// TwinCAT 3 PLC project Untitled1
// ProgramVersion: 3.1.4023.0
// CompilerDefines: VISU_USEWSTRING
// libraries:
//   Tc2_Standard, * (Beckhoff Automation GmbH)
//   Tc2_System, * (Beckhoff Automation GmbH)
//   Tc3_Module, * (Beckhoff Automation GmbH)
//   VisuDialogs, * (System)
//   MachineManage,1.3.1.0,Secote
//   VisuSymbols,3.5.10.0,System
// project tree:
//   DUTs/ E_Axis.TcDUT, E_Cylinder.TcDUT, E_LineAxis.TcDUT, E_LoadClose.TcDUT, E_LoadClass.TcDUT, E_MachineType.TcDUT, E_Timer.TcTLEO, ST_TimeOut.TcDUT, E_ProductType.TcDUT, E_Station.TcDUT, ST_Handshake.TcDUT, ST_Input.TcDUT, ST_Output.TcDUT, ST_Recipe.TcDUT, ST_Setting.TcDUT
//   / GlobalTextList.TcGTLO, PlcTask.TcTTO, RecipeManager.TcRMO (not stored), Version.TcPOU, VISU_TASK.TcTTO, 视图管理器.TcVMO (not stored)
//   GVLs/ GVL.TcGVL, GVL_Data.TcGVL, GVL_IO.TcGVL
//   POUs/Device/ ArrayBool_TO_ArrayByte.TcPOU, ArrayBool_TO_Byte.TcPOU, ArrayByte_TO_ArrayBool.TcPOU, Byte_TO_ArrayBool.TcPOU, FB_LineAxis.TcPOU
//   POUs/ MAIN.TcPOU, P_Alarm.TcPOU, P_Device.TcPOU, P_StationAcquire.TcPOU, P_StationLine1Load.TcPOU, P_StationTakeUc.TcPOU, P_StationLine0Buffer.TcPOU, P_StationLine0Load.TcPOU, P_StationOpenLock.TcPOU, P_StationSteering.TcPOU, P_StationTakeUc_M.TcPOU, P_StationUnloadFrock.TcPOU, P_StationUnloadFrock_L.TcPOU, P_StationUnloadUc_L.TcPOU, P_System.TcPOU
//   VISUs/Ctrl/ CtrlAxisInput.TcVIS, CtrlCylinder_Page.TcVIS, CtrlInput.TcVIS (not stored), CtrlLine.TcVIS, CtrlOther.TcVIS (not stored), CtrlOutput.TcVIS, Cyliner1.TcVIS, Cyliner1_1.TcVIS, Cyliner2.TcVIS, Cyliner3.TcVIS, Cyliner4.TcVIS, Cyliner4_1.TcVIS, Cyliner5.TcVIS, FrameMain.TcVIS, ImagePool.TcIPO (not stored), CtrlPageSetting.TcVIS
//   VISUs/ PageData.TcVIS, PageHome.TcVIS, PageMessage.TcVIS, PageMonitor.TcVIS, PageSetting_AcquireLoad.TcVIS, PageSetting_AcquireLoad_2.TcVIS, PageSetting_OpenLock_2.TcVIS, PageSetting_TakeUc.TcVIS, PageSetting_Steering.TcVIS, PageSetting_Other.TcVIS, PageSetting_Unload_L.TcVIS, PageSetting_OpenLock.TcVIS, PageSetting_UnloadFrock.TcVIS, PageSetting_TakeUc_M.TcVIS, PageSetting.TcVIS
//   VISUs/Text/ InputText.TcTLO, LineLoadClose.TcTLO, LineLoadClase.TcTLO, LoadPriority.TcTLO, MachineType.TcTLO, ProductType.TcTLO, ManualText.TcTLO, OutputText.TcTLO, StationName.TcTLO

CONFIGURATION Untitled1
    RESOURCE PLC ON TwinCAT3
        TASK PlcTask(INTERVAL := T#2ms, PRIORITY := 20);
        TASK VISU_TASK(INTERVAL := T#50000us, PRIORITY := 30);
        PROGRAM MAIN WITH PlcTask : MAIN;
        PROGRAM VisuElems_Visu_Prg WITH VISU_TASK : VisuElems.Visu_Prg;
    END_RESOURCE
END_CONFIGURATION

// ---- DUTs/E_Axis.TcDUT
{attribute 'qualified_only'}
{attribute 'strict'}
TYPE E_Axis :
(
	Z := 1// Z轴
);
END_TYPE

// ---- DUTs/E_Cylinder.TcDUT
{attribute 'qualified_only'}
{attribute 'strict'}
TYPE E_Cylinder :
(
Line0Part:=0, //  主流线分料气缸
Line0Prevent, //  主流线阻挡气缸
Line0Push, //  主流线拨料气缸
AcquirePrevent0, //  接驳线前阻挡气缸
AcquirePrevent1, //  接驳线后阻挡气缸
AcquireLift, //  接驳线顶升气缸
AcquirePush, //  接驳模组拨料气缸
AcquireElevator, //  接驳模组升降气缸
SteeringLift, //  转向站顶升气缸
SteeringAcquireElevator, //  转向站接驳升降气缸
SteeringRotate, //  转向站旋转气缸
SteeringAcquireLimit, //  转向站接驳限位气缸
OpenLockPrevent, //  解锁站阻挡气缸
OpenLockLift, //  解锁站顶升气缸
OpenLockPush, //  解锁站侧推气缸
OpenLockRotate, //  解锁站旋转气缸
OpenLockPush2, //  解锁站侧推气缸2
TakeUcPrevent, //  取UC站阻挡气缸
TakeUcLift, //  取UC站顶升气缸
TakeUcPush, //  取UC站侧推气缸
TakeUcRotate, //  取UC站旋转气缸
TakeUcStandard, //  取UC站校平气缸
UnloadFrockPrevent, //  下工装站阻挡气缸
UnloadFrockLift, //  下工装站顶升气缸
UnloadFrockPush, //  下工装站拨料气缸
TakeUc1Y, //  取UC模组平移Y气缸
TakeUc1Z1, //  取UC模组升降Z1气缸
TakeUc1Z2, //  取UC模组升降Z2气缸
TakeUc1Rotate, //  取UC模组旋转气缸
TakeUc1Clamp, //  取UC模组夹紧气缸
UnloadUcElevator, //  下UC皮带升降气缸
UnloadUcConveyorPush, //  下UC皮带拨料气缸
UnloadFrockConveyorPrevent, //  下工装皮带升降气缸
UnloadFrockConveyorPush, //  下工装皮带拨料气缸
OpenLockElevator,// 解锁站升降气缸
OpenLockPin,// 解锁站压紧气缸
TakeUcElevator,// 取UC站升降气缸
TakeUcPush1,// 取UC站侧推气缸1
UnloadUcBeltTipper,// 下UC皮带翻转
UnloadUcBeltLift,// 下UC皮带顶升
OpenLockTranslation,// 解锁站解锁平移气缸
TakeUcFrockClamp,//取UC站工装夹紧气缸
OpenLockPressPush,//解锁站解压侧推气缸
OpenLockPressRotate,//解锁站解压旋转气缸
AcquirePrevent2,//  接驳线前前阻挡气缸
Line0PushElevator, //  主流线拨料升降气缸
Length
);
END_TYPE

// ---- DUTs/E_LineAxis.TcDUT
{attribute 'qualified_only'}
{attribute 'strict'}
TYPE E_LineAxis :
(
	UnloadUc := 1,// 下Uc线体
	UnloadForck,// 下工装线条
	Acquire,// 接驳站线体
	Dismantling,// 拆解站线体
	AcquireFront // 接驳站前线体
);
END_TYPE

// ---- DUTs/E_LoadClose.TcDUT
{attribute 'qualified_only'}
{attribute 'strict'}
TYPE E_LoadClose :
(
	None:=0,
	Line0,// 关闭Line0
	Acquire// 关闭接驳站上料
);
END_TYPE

// ---- DUTs/E_LoadClass.TcDUT
{attribute 'qualified_only'}
{attribute 'strict'}
TYPE E_LoadClass :
(
	None:=0,
	Line0,// 优先Line0
	Acquire,// 优先接驳站
	Sensor // 优先传感器检测
);
END_TYPE

// ---- DUTs/E_MachineType.TcDUT
{attribute 'qualified_only'}
{attribute 'strict'}
TYPE E_MachineType :
(
	None:=0,
	_367,
	_200,
	_373,
	_069,
	_311
);
END_TYPE

// ---- DUTs/E_Timer.TcTLEO
{attribute 'qualified_only'}
{attribute 'strict'}
TYPE E_Timer :
(
	Timer0 := 0,
	Line0PriorityOnDelay,     // 主流线优先置位延时
	Line0PriorityOffDelay,    // 主流线优先复位延时
	SteeringCheck1F,
	OpenLockCheckF,
	Timer5,
	Timer6,
	Timer7,
	Timer8,
	Timer9,
	Timer10,
	Timer11,
	Timer12,
	Timer13,
	Timer14,
	Timer15,
	Timer16,
	Timer17,
	Timer18,
	Timer19
	
);
END_TYPE

// ---- DUTs/ST_TimeOut.TcDUT
TYPE ST_TimeOut :
STRUCT
	bAcquireCheck2:             BOOL;//接驳线光电检测超时
    bLine0Check3:               BOOL;//主流线到位光电检测超时	
	bOpenLockCheck:             BOOL;//解锁站到位光电检测超时
	bSteeringCheck1:            BOOL;//转向站到位光电检测超时
	bTakeUcCheck1:              BOOL;//取UC站到位光电检测超时
	bUnloadUcCheck1:			BOOL;//翻转气缸到位光电检测超时
	bUnloadFrockCheck1:         BOOL;//下工装站到位光电检测超时
	bUnloadFrockConveyorCheck2: BOOL;//下工装皮带到位光电检测超时
	bUnloadUcCheck2:            BOOL;//下UC皮带到位光电检测超时
	bLine0Check2:               BOOL;//主流线阻挡光电检测超时
	bLine0PushElevatorUp:       BOOL;//主流线拨料升降气缸上升速度过慢
END_STRUCT
END_TYPE

// ---- DUTs/E_ProductType.TcDUT
{attribute 'qualified_only'}
{attribute 'strict'}
TYPE E_ProductType :
(
	None:= 0,
	Left,
	Right
);
END_TYPE

// ---- DUTs/E_Station.TcDUT
{attribute 'qualified_only'}
{attribute 'strict'}
TYPE E_Station :
(
Acquire:=0,//接驳站
Line0Buffer,//主流线缓存
Line0Load,//主流线上料
OpenLock,//解锁站
Steering,//转向站
TakeUc,//取Uc站
TakeUc_M,//取Uc模组
UnloadFrock,//下工装
UnloadFrock_L,//下工装线体
UnloadUc_L,//下UC线体
Line1Load,//接驳线上料
Length
);
END_TYPE

// ---- DUTs/ST_Handshake.TcDUT
TYPE ST_Handshake :
STRUCT
	bBufferToLoad:				BOOL;// 上料缓存站 请求 上料站 放料
	bLoadToBuffer:				BOOL;// 上料站 收到 缓存站请求
	
	bLine1ToAcquire:			BOOL;// 接驳线 请求 接驳站 收料
	bAcquireToLine1:			BOOL;// 接驳站 收到 接驳线请求
	
	bBufferToAcquire:			BOOL;// 上料缓存站 请求 接驳站收料
	bAcquireToBuffer:			BOOL;// 接驳站收 上料缓存站请求
	
	bSteering:					BOOL;// 转向站 请求 放料
	bSteeringOk:				BOOL;// 收到 转向站请求信号
	
	bOpenToSteering:			BOOL;// 解锁站 请求 转向站放料
	bSteeringToOpen:			BOOL;// 转向站 收到 解锁站请求
	
	bTakeUcToOpen:				BOOL;// 取U站 请求 解锁站放料
	bOpenToTakeUc:				BOOL;// 解锁站 收到 取Uc站请求
	
	bTakeUcToTakeUc_M:			BOOL;// 取UC站 请求 取UC模组取料
	bTakeUc_MToTakeUc:			BOOL;// 取Uc模组 收到取Uc站请求
	
	bTakeUcToTakeUc_M_2:			BOOL;// 取UC站 请求 取UC模组取料
	bTakeUc_MToTakeUc_2:			BOOL;// 取Uc模组 收到取Uc站请求
	
	
	bUnloadFrockToTakeUc:		BOOL;//	下工装站 请求 取Uc站放料
	bTakeUcToUnloadFrock:		BOOL;// 取Uc站 收到 下工装站请求
	
	bTakeUc_MToUnloadUcConveyor:BOOL;// 下Uc模组 请求 下Uc线体放料
	bUnloadUcConveyorToTakeUc_M:BOOL;// 下Uc线体 收到 下Uc模组请求
	
	bUnloadFrockToUnloadFrock_L:BOOL;// 下工装站 请求 下工装线体放料
	bUnloadFrock_LToUnloadFrock:BOOL;// 下工装线体 收到 下工装站请求   
END_STRUCT
END_TYPE

// ---- DUTs/ST_Input.TcDUT
TYPE ST_Input :
STRUCT
bStart:BOOL;//启动 IN00
bStop:bool;//停止 IN01
bResetAlarm:bool;//复位 IN02
bEStop:bool;//急停 IN03
bDoor:bool;//安全门开关 IN04
bFrockCloseCheck:BOOL;//工装误合盖检测 IN05
bOpenLockCheck0:BOOL;//解锁站流入光电 IN06
bNone3:bool;//预留 IN07
bLine0PushElevator_Cyl_H:BOOL;//主流线拨料升降气缸原位 IN08
bLine0PushElevator_Cyl_W:BOOL;//主流线拨料升降气缸工作位 IN09
bNone6:bool;//预留 IN0A
bNone7:bool;//预留 IN0B
bLine0Push_Cyl_Safe:BOOL;//主流线拨料气缸安全位 IN0C
bAcquireCheck0:BOOL;//接驳线前阻挡光电 IN0D
bAcquirePrevent2_Cyl_H:BOOL;//接驳线前前阻挡气缸原位 IN0E
bAcquirePrevent2_Cyl_W:BOOL;//接驳线前前阻挡气缸工作位 IN0F
bLine0Part_Cyl_H:bool;//主流线分料气缸原位 IN10
bLine0Part_Cyl_W:bool;//主流线分料气缸工作位 IN11
bLine0Prevent_Cyl_H:bool;//主流线阻挡气缸原位 IN12
bLine0Prevent_Cyl_W:bool;//主流线阻挡气缸工作位 IN13
bLine0Push_Cyl_H:bool;//主流线拨料气缸原位 IN14
bLine0Push_Cyl_W:bool;//主流线拨料气缸工作位 IN15
bAcquirePrevent0_Cyl_H:bool;//接驳线前阻挡气缸原位 IN16
bAcquirePrevent0_Cyl_W:bool;//接驳线前阻挡气缸工作位 IN17
bAcquirePrevent1_Cyl_H:bool;//接驳线后阻挡气缸原位 IN18
bAcquirePrevent1_Cyl_W:bool;//接驳线后阻挡气缸工作位 IN19
bAcquireLift_Cyl_H:bool;//接驳线顶升气缸原位 IN1A
bAcquireLift_Cyl_W:bool;//接驳线顶升气缸工作位 IN1B
bAcquirePush_Cyl_H:bool;//接驳模组拨料气缸原位 IN1C
bAcquirePush_Cyl_W:bool;//接驳模组拨料气缸工作位 IN1D
bAcquireElevator_Cyl_H:bool;//接驳模组升降气缸原位 IN1E
bAcquireElevator_Cyl_W:bool;//接驳模组升降气缸工作位 IN1F
bSteeringLift_Cyl_H:bool;//转向站顶升气缸原位 IN20
bSteeringLift_Cyl_W:bool;//转向站顶升气缸工作位 IN21
bSteeringAcquireElevator_Cyl_H:bool;//转向站接驳升降气缸原位 IN22
bSteeringAcquireElevator_Cyl_W:bool;//转向站接驳升降气缸工作位 IN23
bSteeringRotate_Cyl_H:bool;//转向站旋转气缸原位 IN24
bSteeringRotate_Cyl_W:bool;//转向站旋转气缸工作位 IN25
bSteeringAcquireLimit_Cyl_H:bool;//转向站接驳限位气缸原位 IN26
bSteeringAcquireLimit_Cyl_W:bool;//转向站接驳限位气缸工作位 IN27
bOpenLockPrevent_Cyl_H:bool;//解锁站阻挡气缸原位 IN28
bOpenLockPrevent_Cyl_W:bool;//解锁站阻挡气缸工作位 IN29
bOpenLockLift_Cyl_H:bool;//解锁站顶升气缸原位 IN2A
bOpenLockLift_Cyl_W:bool;//解锁站顶升气缸工作位 IN2B
bOpenLockPush_Cyl_H:bool;//解锁站侧推气缸原位 IN2C
bOpenLockPush_Cyl_W:bool;//解锁站侧推气缸工作位 IN2D
bOpenLockRotate_Cyl_H:bool;//解锁站旋转气缸原位 IN2E
bOpenLockRotate_Cyl_W:bool;//解锁站旋转气缸工作位 IN2F
bOpenLockPush2_Cyl_H:bool;//解锁站侧推气缸2原位 IN30
bOpenLockPush2_Cyl_W:bool;//解锁站侧推气缸2工作位 IN31
bTakeUcPrevent_Cyl_H:bool;//取UC站阻挡气缸原位 IN32
bTakeUcPrevent_Cyl_W:bool;//取UC站阻挡气缸工作位 IN33
bTakeUcLift_Cyl_H:bool;//取UC站顶升气缸原位 IN34
bTakeUcLift_Cyl_W:bool;//取UC站顶升气缸工作位 IN35
bTakeUcPush_Cyl_H:bool;//取UC站侧推气缸原位 IN36
bTakeUcPush_Cyl_W:bool;//取UC站侧推气缸工作位 IN37
bTakeUcRotate_Cyl_H:bool;//取UC站旋转气缸原位 IN38
bTakeUcRotate_Cyl_W:bool;//取UC站旋转气缸工作位 IN39
bTakeUcStandard_Cyl_H:bool;//取UC站校平气缸原位 IN3A
bTakeUcStandard_Cyl_W:bool;//取UC站校平气缸工作位 IN3B
bTakeUcFrockClamp_Cyl_H:BOOL;//取UC站工装夹紧气缸原位 IN3C
bTakeUcFrockClamp_Cyl_W:BOOL;//取UC站工装夹紧气缸工作位 IN3D
bUnloadFrockPrevent_Cyl_H:bool;//下工装站阻挡气缸原位 IN3E
bUnloadFrockPrevent_Cyl_W:bool;//下工装站阻挡气缸工作位 IN3F
bUnloadFrockLift_Cyl_H:bool;//下工装站顶升气缸原位 IN40
bUnloadFrockLift_Cyl_W:bool;//下工装站顶升气缸工作位 IN41
bUnloadFrockPush_Cyl_H:bool;//下工装站拨料气缸原位 IN42
bUnloadFrockPush_Cyl_W:bool;//下工装站拨料气缸工作位 IN43
bTakeUc1Y_Cyl_H:bool;//取UC模组平移Y气缸原位 IN44
bTakeUc1Y_Cyl_W:bool;//取UC模组平移Y气缸工作位 IN45
bTakeUc1Z1_Cyl_H:bool;//取UC模组升降Z1气缸原位 IN46
bTakeUc1Z1_Cyl_W:bool;//取UC模组升降Z1气缸工作位 IN47
bTakeUc1Z2_Cyl_H:bool;//取UC模组升降Z2气缸原位 IN48
bTakeUc1Z2_Cyl_W:bool;//取UC模组升降Z2气缸工作位 IN49
bTakeUc1Rotate_Cyl_H:bool;//取UC模组旋转气缸原位 IN4A
bTakeUc1Rotate_Cyl_W:bool;//取UC模组旋转气缸工作位 IN4B
bTakeUc1Clamp_Cyl_H:bool;//取UC模组夹紧气缸原位 IN4C
bTakeUc1Clamp_Cyl_W:bool;//取UC模组夹紧气缸工作位 IN4D
bUnloadUcElevator_Cyl_H:bool;//下UC皮带升降气缸原位 IN4E
bUnloadUcElevator_Cyl_W:bool;//下UC皮带升降气缸工作位 IN4F
bUnloadUcConveyorPush_Cyl_H:bool;//下UC皮带拨料气缸原位 IN50
bUnloadUcConveyorPush_Cyl_W:bool;//下UC皮带拨料气缸工作位 IN51
bUnloadFrockConveyorPrevent_Cyl_H:bool;//下工装皮带升降气缸原位 IN52
bUnloadFrockConveyorPrevent_Cyl_W:bool;//下工装皮带升降气缸工作位 IN53
bUnloadFrockConveyorPush_Cyl_H:bool;//下工装皮带拨料气缸原位 IN54
bUnloadFrockConveyorPush_Cyl_W:bool;//下工装皮带拨料气缸工作位 IN55
bOpenLockPressPush_Cyl_H:BOOL;//解锁站解压侧推气缸原位 IN56
bOpenLockPressPush_Cyl_W:BOOL;//解锁站解压侧推气缸工作位 IN57
bOpenLockPressRotate_Cyl_H:BOOL;//解锁站解压旋转气缸原位 IN58
bOpenLockPressRotate_Cyl_W:BOOL;//解锁站解压旋转气缸工作位 IN59
bNone34:bool;//预留 IN5A
bNone35:bool;//预留 IN5B
bUnloadUcBeltTipper_Cyl_H:bool;//下UC皮带翻转气缸缩回 IN5C
bUnloadUcBeltTipper_Cyl_W:bool;//下UC皮带翻转气缸伸出 IN5D
bUnloadUcBeltLift_Cyl_H:bool;//下UC皮带顶升气缸缩回 IN5E
bUnloadUcBeltLift_Cyl_W:bool;//下UC皮带顶升气缸伸出 IN5F
bLine0Check1:bool;//主流线分料光电 IN60
bLine0Check2:bool;//主流线阻挡光电 IN61
bLine0Check3:bool;//主流线到位光电 IN62
bAcquireCheck1:bool;//接驳线流入光电 IN63
bAcquireCheck2:bool;//接驳线到位光电 IN64
bSteeringCheck1:bool;//转向站到位光电 IN65
bOpenLockCheck:bool;//解锁站到位光电 IN66
bTakeUcCheck1:bool;//取UC站到位光电 IN67
bUnloadFrockCheck1:bool;//下工装站到位光电 IN68
bUnloadUcCheck1:bool;//下UC皮带流入光电 IN69
bUnloadUcCheck2:bool;//下UC皮带到位光电 IN6A
bUnloadFrockCheck0:BOOL;//下工装站流入光电 IN6B
bUnloadFrockConveyorCheck2:bool;//下工装皮带到位光电 IN6C
bUnloadUcBeltTipper:bool;//下uc皮带翻转光电 IN6D
bTakeUcCheck0:BOOL;//取UC站流入光电 IN6E
bTakeUc1Y_Cyl_Safe:BOOL;//取UC模组平移Y气缸安全位 IN6F
bOpenLockElevator_Cyl_H:bool;//解锁站升降气缸原位 IN70
bOpenLockElevator_Cyl_W:bool;//解锁站升降气缸工作位 IN71
bOpenLockTranslation_Cyl_H:bool;//解锁站解锁平移原位 IN72
bOpenLockTranslation_Cyl_W:bool;//解锁站解锁平移工作位 IN73
bOpenLockPin_Cyl_H:bool;//解锁站按压气缸到原位 IN74
bOpenLockPin_Cyl_W:bool;//解锁站按压气缸到工作位 IN75
bTakeUcElevator_Cyl_H:bool;//取UC站升降气缸原位 IN76
bTakeUcElevator_Cyl_W:bool;//取UC站升降气缸工作位 IN77
bTakeUcPush1_Cyl_H:bool;//取UC站侧推1气缸到原位 IN78
bTakeUcPush1_Cyl_W:bool;//取UC站侧推1气缸到工作位 IN79
bNone45:bool;//预留 IN7A
bNone46:bool;//预留 IN7B
bNone47:bool;//预留 IN7C
bNone48:bool;//预留 IN7D
bNone49:bool;//预留 IN7E
bNone50:bool;//预留 IN7F

END_STRUCT
END_TYPE

// ---- DUTs/ST_Output.TcDUT
TYPE ST_Output :
STRUCT
bBeacon_Red:BOOL;//三色灯红 OUT00
bBeacon_Yellow:bool;//三色灯黄 OUT01
bBeacon_Green:bool;//三色灯绿 OUT02
bBeacon_Buzzer:bool;//蜂鸣器 OUT03
bRuning:bool;//运行指示灯 OUT04
bStop:bool;//停止指示灯 OUT05
bLED:bool;//照明灯 OUT06
bNone1:bool;//预留 OUT07
bOpenLockPressPush_Cyl_H:BOOL;//解锁站解压侧推气缸到原位 OUT08
bOpenLockPressPush_Cyl_W:BOOL;//解锁站解压侧推气缸到工作位 OUT09
bOpenLockPressRotate_Cyl_H:BOOL;//解锁站解压旋转气缸到原位 OUT0A
bOpenLockPressRotate_Cyl_W:BOOL;//解锁站解压旋转气缸到工作位 OUT0B
bLine0PushElevator_Cyl_H:BOOL;//主流线拨料升降气缸到原位 OUT0C
bLine0PushElevator_Cyl_W:BOOL;//主流线拨料升降气缸到工作位 OUT0D
bAcquirePrevent2_Cyl_H:BOOL;//接驳线前前阻挡气缸缩回 OUT0E
bAcquirePrevent2_Cyl_W:BOOL;//接驳线前前阻挡气缸伸出 OUT0F
bLine0Part_Cyl_H:bool;//主流线分料气缸缩回 OUT10
bLine0Part_Cyl_W:bool;//主流线分料气缸伸出 OUT11
bLine0Prevent_Cyl_H:bool;//主流线阻挡气缸缩回 OUT12
bLine0Prevent_Cyl_W:bool;//主流线阻挡气缸伸出 OUT13
bLine0Push_Cyl_H:bool;//主流线拨料气缸缩回 OUT14
bLine0Push_Cyl_W:bool;//主流线拨料气缸伸出 OUT15
bAcquirePrevent0_Cyl_H:bool;//接驳线前阻挡气缸缩回 OUT16
bAcquirePrevent0_Cyl_W:bool;//接驳线前阻挡气缸伸出 OUT17
bAcquirePrevent1_Cyl_H:bool;//接驳线后阻挡气缸缩回 OUT18
bAcquirePrevent1_Cyl_W:bool;//接驳线后阻挡气缸伸出 OUT19
bAcquireLift_Cyl_H:bool;//接驳线顶升气缸缩回 OUT1A
bAcquireLift_Cyl_W:bool;//接驳线顶升气缸伸出 OUT1B
bAcquirePush_Cyl_H:bool;//接驳模组拨料气缸缩回 OUT1C
bAcquirePush_Cyl_W:bool;//接驳模组拨料气缸伸出 OUT1D
bAcquireElevator_Cyl_H:bool;//接驳模组升降气缸缩回 OUT1E
bAcquireElevator_Cyl_W:bool;//接驳模组升降气缸伸出 OUT1F
bSteeringLift_Cyl_H:bool;//转向站顶升气缸缩回 OUT20
bSteeringLift_Cyl_W:bool;//转向站顶升气缸伸出 OUT21
bSteeringAcquireElevator_Cyl_H:bool;//转向站接驳升降气缸缩回 OUT22
bSteeringAcquireElevator_Cyl_W:bool;//转向站接驳升降气缸伸出 OUT23
bSteeringRotate_Cyl_H:bool;//转向站旋转气缸缩回 OUT24
bSteeringRotate_Cyl_W:bool;//转向站旋转气缸伸出 OUT25
bSteeringAcquireLimit_Cyl_H:bool;//转向站接驳限位气缸缩回 OUT26
bSteeringAcquireLimit_Cyl_W:bool;//转向站接驳限位气缸伸出 OUT27
bOpenLockPrevent_Cyl_H:bool;//解锁站阻挡气缸缩回 OUT28
bOpenLockPrevent_Cyl_W:bool;//解锁站阻挡气缸伸出 OUT29
bOpenLockLift_Cyl_H:bool;//解锁站顶升气缸缩回 OUT2A
bOpenLockLift_Cyl_W:bool;//解锁站顶升气缸伸出 OUT2B
bOpenLockPush_Cyl_H:bool;//解锁站侧推气缸缩回 OUT2C
bOpenLockPush_Cyl_W:bool;//解锁站侧推气缸伸出 OUT2D
bOpenLockRotate_Cyl_H:bool;//解锁站旋转气缸缩回 OUT2E
bOpenLockRotate_Cyl_W:bool;//解锁站旋转气缸伸出 OUT2F
bOpenLockPush2_Cyl_H:bool;//解锁站侧推气缸2缩回 OUT30
bOpenLockPush2_Cyl_W:bool;//解锁站侧推气缸2伸出 OUT31
bTakeUcPrevent_Cyl_H:bool;//取UC站阻挡气缸缩回 OUT32
bTakeUcPrevent_Cyl_W:bool;//取UC站阻挡气缸伸出 OUT33
bTakeUcLift_Cyl_H:bool;//取UC站顶升气缸缩回 OUT34
bTakeUcLift_Cyl_W:bool;//取UC站顶升气缸伸出 OUT35
bTakeUcPush_Cyl_H:bool;//取UC站侧推气缸缩回 OUT36
bTakeUcPush_Cyl_W:bool;//取UC站侧推气缸伸出 OUT37
bTakeUcRotate_Cyl_H:bool;//取UC站旋转气缸缩回 OUT38
bTakeUcRotate_Cyl_W:bool;//取UC站旋转气缸伸出 OUT39
bTakeUcStandard_Cyl_H:bool;//取UC站校平气缸原位 OUT3A
bTakeUcStandard_Cyl_W:bool;//取UC站校平气缸工作位 OUT3B
bTakeUcFrockClamp_Cyl_H:BOOL;//取UC站工装夹紧气缸原位 OUT3C
bTakeUcFrockClamp_Cyl_W:bool;//取UC站工装夹紧气缸工作位 OUT3D
bUnloadFrockPrevent_Cyl_H:BOOL;//下工装站阻挡气缸缩回 OUT3E
bUnloadFrockPrevent_Cyl_W:bool;//下工装站阻挡气缸伸出 OUT3F
bUnloadFrockLift_Cyl_H:bool;//下工装站顶升气缸缩回 OUT40
bUnloadFrockLift_Cyl_W:bool;//下工装站顶升气缸伸出 OUT41
bUnloadFrockPush_Cyl_H:bool;//下工装站拨料气缸缩回 OUT42
bUnloadFrockPush_Cyl_W:bool;//下工装站拨料气缸伸出 OUT43
bTakeUc1Y_Cyl_H:bool;//取UC模组平移Y气缸缩回 OUT44
bTakeUc1Y_Cyl_W:bool;//取UC模组平移Y气缸伸出 OUT45
bTakeUc1Z1_Cyl_H:bool;//取UC模组升降Z1气缸缩回 OUT46
bTakeUc1Z1_Cyl_W:bool;//取UC模组升降Z1气缸伸出 OUT47
bTakeUc1Z2_Cyl_H:bool;//取UC模组升降Z2气缸缩回 OUT48
bTakeUc1Z2_Cyl_W:bool;//取UC模组升降Z2气缸伸出 OUT49
bTakeUc1Rotate_Cyl_H:bool;//取UC模组旋转气缸缩回 OUT4A
bTakeUc1Rotate_Cyl_W:bool;//取UC模组旋转气缸伸出 OUT4B
bTakeUc1Clamp_Cyl_H:bool;//取UC模组夹紧气缸缩回 OUT4C
bTakeUc1Clamp_Cyl_W:bool;//取UC模组夹紧气缸伸出 OUT4D
bUnloadUcElevator_Cyl_H:bool;//下UC皮带升降气缸缩回 OUT4E
bUnloadUcElevator_Cyl_W:bool;//下UC皮带升降气缸伸出 OUT4F
bUnloadUcConveyorPush_Cyl_H:bool;//下UC皮带拨料气缸缩回 OUT50
bUnloadUcConveyorPush_Cyl_W:bool;//下UC皮带拨料气缸伸出 OUT51
bUnloadFrockConveyorPrevent_Cyl_H:bool;//下工装皮带升降气缸缩回 OUT52
bUnloadFrockConveyorPrevent_Cyl_W:bool;//下工装皮带升降气缸伸出 OUT53
bUnloadFrockConveyorPush_Cyl_H:bool;//下工装皮带拨料气缸缩回 OUT54
bUnloadFrockConveyorPush_Cyl_W:bool;//下工装皮带拨料气缸伸出 OUT55
bAcquireFrontAxis:BOOL;//接驳站前步进 OUT56
bAcquireAxis:bool;//接驳线步进 OUT57
bDismantlingAxis:bool;//拆解线步进 OUT58
bUnloadUcAxis:bool;//下UC皮带步进 OUT59
bUnloadFrock:bool;//下工装皮带步进 OUT5A
bNone21:bool;//预留 OUT5B
bUnloadUcBeltTipper_Cyl_H:bool;//下UC皮带翻转气缸缩回 OUT5C
bUnloadUcBeltTipper_Cyl_W:bool;//下UC皮带翻转气缸伸出 OUT5D
bUnloadUcBeltLift_Cyl_H:bool;//下UC皮带顶升气缸缩回 OUT5E
bUnloadUcBeltLift_Cyl_W:bool;//下UC皮带顶升气缸伸出 OUT5F
bOpenLockElevator_Cyl_H:bool;//解锁站升降气缸原位 OUT60
bOpenLockElevator_Cyl_W:bool;//解锁站升降气缸工作位 OUT61
bOpenLockTranslation_Cyl_H:bool;//解锁站解锁平移原位 OUT62
bOpenLockTranslation_Cyl_W:bool;//解锁站解锁平移工作位 OUT63
bOpenLockPin_Cyl_H:bool;//解锁站按压气缸到原位 OUT64
bOpenLockPin_Cyl_W:bool;//解锁站按压气缸到工作位 OUT65
bTakeUcElevator_Cyl_H:bool;//取UC站升降气缸原位 OUT66
bTakeUcElevator_Cyl_W:bool;//取UC站升降气缸工作位 OUT67
bTakeUcPush1_Cyl_H:bool;//取UC站侧推1气缸到原位 OUT68
bTakeUcPush1_Cyl_W:bool;//取UC站侧推1气缸到工作位 OUT69
bNone35:BOOL;//预留 OUT6A
bNone36:BOOL;//预留 OUT6B
bNone37:BOOL;//预留 OUT6C
bNone38:BOOL;//预留 OUT6D
bNone39:bool;//预留 OUT6E
bNone40:bool;//预留 OUT6F

END_STRUCT
END_TYPE

// ---- DUTs/ST_Recipe.TcDUT
TYPE ST_Recipe :
STRUCT
	arrInputTon:				ARRAY[0..7,0..15] OF UINT;
	arrOutputTon:				ARRAY[0..6,0..15] OF UINT;
	arrAutoTon:				    ARRAY[0..19] OF UINT;	
	
	eMachineType:				E_MachineType;
	eProductType:               E_ProductType;//产品类型（左，右）
	eLoadClass:					E_LoadClass;
	eLoadClose:					E_LoadClose;
	
	bLuxshardict:				BOOL;
END_STRUCT
END_TYPE

// ---- DUTs/ST_Setting.TcDUT
TYPE ST_Setting :
STRUCT
	bDryRun:					BOOL;// 空跑
	bManualLoad:				BOOL;// 手动上料
	bManualUnloadUc:			BOOL;// 手动下UC
	bManualUnloadFrock:			BOOL;// 手动下工装
	arrStationShield:			ARRAY[0..20] OF BOOL;// 工站使能信号
	bLine0BufferShield:         BOOL;// 主流分料屏蔽
	bSafeDoorShield:            BOOL;// 安全门屏蔽
	bOpenLockPressShield:       BOOL;// 解锁站解除保压屏蔽
	bAcquirePrevent2Shield:     BOOL;// 接驳线前前阻挡气缸屏蔽
	bStopFrontStation:          BOOL;// 不允许前站放料
	bLine0Priority:             BOOL;// 优先主流线上料
	bFrockCloseCheckShield:     BOOL;// 工装误合盖检测屏蔽
END_STRUCT
END_TYPE

// ---- GVLs/GVL.TcGVL
{attribute 'qualified_only'}
VAR_GLOBAL
	I:					ST_Input;
	Q:					ST_Output;
	stSetting:			ST_Setting;// 设置参数
	
	stShield_I:			ARRAY[0..7,0..15] OF  BOOL;
	stShield_Q:			ARRAY[0..6,0..15] OF  BOOL;
	
	stHandshake:		ST_Handshake;
				
	arrFbLine:			ARRAY[0..10] OF FB_LineAxis;// 流线控制
	
    stOverTime:			ST_TimeOut;//光电超时报警 
	
	_arrAutoTimer:		ARRAY[0..19] OF  TON;//自动流程延时 
	_arrAutoTimerOut:	ARRAY[0..19] OF  BOOL;//自动流程延时输出
	
	TakeUcSafeCheckNG_OpenLock:  BOOL;	//解锁站工装误合盖检测NG记忆
	TakeUcSafeCheckNG_TakeUc:  BOOL;    //取UC站读取解锁站工装误合盖检测NG记忆
	AlarmResetMark:     BOOL;           //311机型主流线拨料升降气缸上升速度过慢报警复位标记
	
END_VAR

// ---- GVLs/GVL_Data.TcGVL
{attribute 'qualified_only'}
VAR_GLOBAL PERSISTENT
	stRecipe:					ST_Recipe;// 配方文件
END_VAR

// ---- GVLs/GVL_IO.TcGVL
{attribute 'qualified_only'}
VAR_GLOBAL
	I_Temp :				ARRAY[0..7,0..15] OF  BOOL;//由绝对点位的字节数组 转化成的布尔数组
	Q_Temp :				ARRAY[0..6,0..15] OF  BOOL;//由绝对点位的字节数组 转化成的布尔数组
	
	I AT %I*:				ARRAY[0..15] OF BYTE;//绝对点位 输入
	Q AT %Q*:				ARRAY[0..13] OF BYTE;//绝对点位 输出

	EIP_I_ConnState AT %I*:				UDINT;// 输入
	EIP_I_Var4090   AT %I*:				WORD;// 输入	
	EIP_Q_ConnCtrl  AT %Q*:				UDINT;// 输出
	EIP_Q_Var4091   AT %Q*:				WORD;// 输出	
	
	
	AxisInput AT %I*:		UDINT;			
END_VAR

// ---- POUs/MAIN.TcPOU
PROGRAM MAIN
VAR
	VERSION:STRING;
END_VAR

GVL_Data.stRecipe.bLuxshardict:=TRUE;

VERSION:='5.5.0';
P_System();
P_Alarm();
P_Device();

P_StationAcquire();// 接驳站
P_StationLine0Buffer();// Line0上料缓存站
P_StationLine0Load();// Line0上料站
P_StationOpenLock();// 解锁站
P_StationSteering();// 转向站
P_StationTakeUc();// 取UC
P_StationTakeUc_M();// 取UC模组
P_StationUnloadFrock();// 下工装
P_StationUnloadFrock_L();// 下工装线条
P_StationUnloadUc_L();// 下UC线条
P_StationLine1Load();// Line1上料站


IF GVL_Data.stRecipe.eMachineType=E_MachineType._367 THEN
	GVL_IO.EIP_Q_Var4091.1:=GVL_P.G_stSystem.stMode.bAutoRunning AND NOT GVL.I.bLine0Check1 AND  NOT GVL.stSetting.bStopFrontStation;//给前站设备要料信号
ELSE
	GVL_IO.EIP_Q_Var4091.1:=GVL_P.G_stSystem.stMode.bAutoRunning AND NOT GVL.I.bAcquireCheck0 AND  NOT GVL.stSetting.bStopFrontStation;//给前站设备要料信号
END_IF

END_PROGRAM

// ---- Version.TcPOU
PROGRAM Version
VAR
END_VAR

//	版本号		修改人		修改日期		修改内容
//	1.2.0		李天		2021.06.27		311空跑后优化373解锁校平气缸
//	1.3.0		李天		2021.06.27		添加下工装阻挡气缸判断
//  1.4.0      刘雪峰       2021.06.28      添加下工装阻挡气缸屏蔽，优化气缸屏蔽，增加气缸空跑程序的调用选择
//  1.5.0      刘雪峰       2021.06.28      添加轴命名，添加取UC模组升降Z2气缸IO屏蔽，增加版本号界面显示，完善转向站和取uc模组流程，增加取uc模组z1z2气缸控制方法调用的判断,完善各机型气缸空跑程序
//  2.0.0      刘雪峰       2021.06.29      更新IO,气缸、轴excel,新增取UC工装夹紧气缸和IO,更新input和output结构体,更新E_cycliner枚举变量,按照机型屏蔽新增的气缸和IO,更新input和output的Textlist,优化取UC工站和取UC模组工站流程,完善正常模式下调用的A_Cylinder程序
//  2.1.0      刘雪峰       2021.07.01      更新气缸调试部分的界面程序，增加产品类型选择，优化转向站和下UC线体流程，添加取UC模组夹紧气缸工作位和解锁站侧推气缸2初始位在空跑时的屏蔽
//	2.2.0		李天		2021.07.02		修改373解锁校平气缸2动作,该气缸只需一直伸出即可;
//  2.2.1      刘雪峰       2021.07.05      修改部分气缸的界面调试控件，优化转向站初始化气缸动作流程；
//  2.3.0       王恒        2021.07.14      增加拨料站（Switch）和翻转站（Tipper）,将接驳模组拨料气缸和接驳模组升降气缸单独组成拨料站，将下UC皮带翻转气缸和下UC皮带顶升气缸单独组成翻转站;
//  2.3.1       王恒        2021.07.23      增加各工站到位光电检测超时报警;增加气缸界面按工站分页功能;主界面增加界面CT显示;增加生产计数显示;增加各到位光电信号显示;增加从转向站手动上料和从下UC、下工装皮带末端手动下料功能；增加屏蔽取UC模组功能，使投入工装时，只验证解锁与扣合，不验证夹取UC动作；
//                                          增加初始化检测各工站光电是否检测有料功能，并在初始化结束添加再次提醒操作员人工检查的5级报警;201机型下UC皮带流入光电IN6B代替下UC皮带翻转光电IN6D,用来检测UC是否到位，下UC皮带翻转光电IN6D不再使用；因为取UC模组Z1气缸上升速度较慢，所以下调了取UC模组Z1气缸的上限位，使Z1气缸的行程尽可能减少;
//  2.3.2       李天        2021.07.25      增加伺服轴持续接触极限报警，无法点动脱离问题，增加相应指示灯和复位功能；
//	2.4.0		李天		2021.07.26		将王恒新增的两个工站（接驳模组站及下UC线体旋转站） 再改回去
//	2.5.0		李天		2021.07.26		在RH069中待料测试 并修改一些细节 不影响整体流程
//	2.5.1		李天		2021.07.27		将手动下UC 手动下工装 手动上料 开放到界面
//	2.5.2		李天		2021.07.27		将报警显示控件放大
//	2.6.0		李天		2021.07.27		修改手动上料跳转空步号问题
//	2.6.1		李天		2021.07.28		添加用户权限 用户名：Admin 密码：333
//	2.6.2		李伟3		2021.07.28		优化201取UC站侧推气缸动作 可提前推出
//	2.7.0		李天		2021.07.31		将下UC流线及下工装流线到位光电报警等级改成3级
//	2.7.1		李伟3		2021.08.2		将自动流程中1471步中取UC模组平移Y气缸硬件IO修改为气缸功能块状态位
//	3.0.0		李伟3		2021.08.3		1.将自动流程中1471步中取UC模组平移Y气缸气缸功能块状态位修改为硬件IO
//                                          2.暂时取消手动页面权限管理，方便调试
//                                          3.将IO监控页面IN6B下工装线体流入光电变更为下工装流线流入光电
//                                          4.修改取UC模组自动程序，添加分支:设备机型为311时，取UC旋转气缸不旋转放料
//                                          5.将设备内工位检测到位光电传感器超时报警由五级报警提升为三级报警，并修复报警无法复位问题
//                                          6.添加 IN6F取UC模组平移Y气缸安全位 传感器,并修改动作流程
//                                          7.修改和优化了311机型设备 取UC站&取UC模组 的自动动作流程,缩短CT时间
//                                          8.在自动程序中添加 下UC线体到位检测超时 报警
//	3.0.1		李伟3		2021.08.5		1.屏蔽画面中添加屏蔽主流线分料气缸的功能
//                                          2.将主画面计数清零按钮增加用户权限
//                                          3.优化修改367机型 取UC模组 自动流程,缩短CT
//                                          4.优化画面按钮相关中文显示
//                                          5.修复了下工装站初始化撞机的问题
//	3.0.2		李伟3		2021.08.6		1.屏蔽画面中添加 蜂鸣器屏蔽 和 安全门屏蔽 的功能
//                                          2.增加 设备运行中安全门被打开 报警
//	4.0.0		李伟3		2021.08.12		1.373机型解锁站增加两个气缸，增加手动&自动&初始化程序
//                                          2.修复373机型手动画面校平气缸未屏蔽的问题
//                                          3.修复373机型IO画面未使用IO点没有屏蔽的问题
//                                          4.修复设备蜂鸣器响声不正常的问题
//                                          5.优化367机型取UC站的自动流程
//	4.1.0		李伟3		2021.08.13		1.增加接驳线阻挡气缸&接驳线光电传感器，增加手动&自动&初始化程序
//	4.1.1		李伟3		2021.08.16		1.优化不同机型手动页面&IO监控页面的显示问题
//	4.2.0		李伟3		2021.08.24		1.将新加的接驳站前流水线由急停按钮控制改为继电器控制，增加手自动程序
//	4.2.1		李伟3		2021.08.25		1.优化201机型下UC皮带翻转顶升气缸动作流程，先让顶升气缸上升再放UC，防止损伤排线
//	4.2.2		李伟3		2021.08.31		1.优化主流线分料气缸和阻挡气缸的动作逻辑,修改主流线分料气缸缩回端为原位,增加主流线阻挡光电检测超时报警
//	4.3.0		李伟3		2021.09.02		1.367机型增加主流线拨料升降气缸，修改手自动程序及画面
//                                          2.修改取UC站初始化动作流程，修复367机型取UC站初始化异常的问题
//	5.0.0		李伟3		2021.09.07		1.增加通过EIP与前站信号交互的配置和程序
//                                          2.修改主流线到位光电检测超时时间为20S,因为主流线速度过慢会误引发报警
//	5.1.0		李伟3		2021.09.10		1.优化了主流线和接驳线上料优先级选择部分的程序，画面上增加了优先级下拉菜单选择
//                                          2.画面上增加了停止前站放料的按钮
//                                          3.增加 主流线拨料气缸安全位 IN0C 传感器，优化367主流线上料流程
//                                          4.增加主流线与接驳线上料优先级根据传感器自动切换逻辑
//                                          5.优化与前站交互要料逻辑
//	5.2.0		李伟3		2021.09.16		1.311机型增加检测工装误合盖传感器，修改动作流程及画面
//                                          2.367机型增加解锁站流入光电传感器，优化动作流程，缩短CT
//                                          3.373机型增加取UC站流入光电传感器，优化动作流程，缩短CT
//                                          4.373机型增加主流线传感器,优化367机型主流线拨料气缸动作，增加主流线拨料升降气缸上升速度过慢报警，防止损伤产品
//                                          5.优化自动程序中所使用的延时，画面上增加延时时间设置
//                                          6.将打开安全门由一级报警修改为3级报警，方便维护
//                                          7.修复取UC站初始化时与取UC模组撞机的问题
//	5.3.0		李伟3		2021.09.17		1.373机型取UC站增加检测工装误合盖传感器，修改动作流程及画面
//	5.4.0		李伟3		2021.09.17		1.修改解锁站和取UC站的放料逻辑，缩短CT
//	5.5.0		李伟3		2021.09.17		1.将接驳站分料气缸和阻挡气缸分离为单独工站，优化交互逻辑

END_PROGRAM

// ---- POUs/P_System.TcPOU
PROGRAM P_System
VAR
	_arrFbButton:			ARRAY[0..10] OF FB_Button;
	_arrTon:				ARRAY[0..10] OF TON;
	_fbCT:					FB_CycleTime1;
	_cttime:				REAL;
	
	_rTRIG:					R_TRIG;
	_iProductionCount:      INT;//产能计数
	_bCountZero:			BOOL;//产能计数清零
END_VAR

A_Machine();
A_System();

ACTION A_Machine:
//CT测试
_fbCT(Execute:=G_arrCylinder[E_Cylinder.TakeUcLift].stOutput.bWork, CycleTime=> );
_cttime:=TIME_TO_REAL(_fbCT.CycleTime)/1000;
//复位 退出空跑模式
IF G_stSystem.stInput.bReset THEN
	GVL.stSetting.bDryRun:=FALSE;
END_IF

//产能计数
_rTRIG(CLK:= G_arrCylinder[E_Cylinder.OpenLockLift].stOutput.bWork, Q=> );
IF G_stSystem.stMode.bAutoRunning AND NOT GVL.stSetting.bDryRun AND _rTRIG.Q THEN
	_iProductionCount:=_iProductionCount+1;
END_IF
IF NOT G_stSystem.stMode.bAutoRunning  AND  _bCountZero THEN
	_iProductionCount:=0;
END_IF
END_ACTION

ACTION A_System:
G_stSystem.stInput.bEStop:=NOT GVL.I.bEStop;
_arrTon[0](IN:=GVL.I.bResetAlarm,PT:=T#3S , Q=>G_stSystem.stInput.bInit , ET=> );


GVL.Q.bBeacon_Buzzer:=G_stSystem.stOutput.bLightRed AND NOT MachineManage.G_stSystem.stInput.bQuiet;
GVL.Q.bRuning:=GVL.Q.bBeacon_Green:=G_stSystem.stOutput.bLightGreen;
GVL.Q.bStop:=GVL.Q.bBeacon_Red:=G_stSystem.stOutput.bLightRed;
GVL.Q.bBeacon_Yellow:=G_stSystem.stOutput.bLightYellow;

_arrFbButton[0](In:=G_stSystem.stInput.bStart, CLK:=GVL.I.bStart );
_arrFbButton[1](In:= G_stSystem.stInput.bStop, CLK:=GVL.I.bStop );
_arrFbButton[2](In:=G_stSystem.stInput.bResetAlarm , CLK:= GVL.I.bResetAlarm  );

G_stSystem.stLogConfig.bExecute:=TRUE;
G_stSystem.stLogConfig.sFilePath:='D:\PLC\Log\System';

P_Machine(StationCount:=E_Station.Length);
END_ACTION

END_PROGRAM

// ---- POUs/P_Alarm.TcPOU
PROGRAM P_Alarm
VAR
	_arrFbErrorTag1:				ARRAY[0..20] OF  FB_ErrorTag;
	_arrFbErrorTag2:				ARRAY[0..20] OF  FB_ErrorTag;
	_arrFbErrorTag3:				ARRAY[0..20] OF  FB_ErrorTag;
	_arrFbErrorTag4:				ARRAY[0..20] OF  FB_ErrorTag;
	_arrFbErrorTag5:				ARRAY[0..20] OF  FB_ErrorTag;
	
	_i:								INT;
	
	_bFirstRun:						BOOL:=true;
END_VAR

G_stError.bSaveLog:=TRUE;
G_stError.sFileLogPath:='D:\PLC\Log\Error';

A_Alarm1();
A_Alarm2();
A_Alarm3();
A_Alarm4();
A_Alarm5();

ACTION A_Alarm1:

_i:=0;
_arrFbErrorTag1[_i].Enable:=NOT GVL.I.bEStop;
_arrFbErrorTag1[_i].Language[E_Language.Chinese]:="急停被按下";


_i:=1;
_arrFbErrorTag1[_i].Enable:=GVL_Data.stRecipe.eMachineType=E_MachineType.None;
_arrFbErrorTag1[_i].Language[E_Language.Chinese]:="设备类型未选择";

_i:=2;
_arrFbErrorTag1[_i].Enable:=GVL_Data.stRecipe.eProductType=E_ProductType.None;
_arrFbErrorTag1[_i].Language[E_Language.Chinese]:="产品类型未选择";



FOR _i:=0 TO 20 BY 1 DO
_arrFbErrorTag1[_i](
	System:=G_stSystem , 
	Error:=G_stError , 
	ID:=TO_BYTE(_i+50) , 
	Category:=E_ErrorCategory.Safety , 
	InfoIndex:= , 
	Enable:= , 
	Message:= , 
	Level:=1 , 
	Position:="P_Alarm:A_Alarm1" , 
	ErrorTime:= , 
	Language:= , 
	Erroring=> , 
	ErrorCode=> );
END_FOR
END_ACTION

ACTION A_Alarm2:
_i:=0;
_arrFbErrorTag2[_i].Enable:=G_arrCylinder[E_Cylinder.TakeUc1Clamp].stOutput.bWork AND NOT G_stSystem.stMode.bHomeDone;
_arrFbErrorTag2[_i].Language[E_Language.Chinese]:="请将夹紧气缸松开后再初始化";


FOR _i:=0 TO 20 BY 1 DO
_arrFbErrorTag2[_i](
	System:=G_stSystem , 
	Error:=G_stError , 
	ID:=TO_BYTE(52) , 
	Category:=E_ErrorCategory.Other , 
	InfoIndex:=TO_BYTE(_i) , 
	Enable:= , 
	Message:= , 
	Level:=2 , 
	Position:="P_Alarm:A_Alarm2" , 
	ErrorTime:= , 
	Language:= , 
	Erroring=> , 
	ErrorCode=> );
END_FOR
END_ACTION

ACTION A_Alarm3:
_i:=0;
_arrFbErrorTag3[_i].Enable:=(G_stSystem.stMode.bHomeDone AND G_arrStation[E_Station.OpenLock].iStepNow = 1000) 
AND (GVL_IO.I_Temp[6,4](*接驳线到位光电*) OR GVL_IO.I_Temp[6,2](*主流线到位光电*) OR GVL_IO.I_Temp[6,6](*解锁站到位光电*) OR 
GVL_IO.I_Temp[6,5](*转向站到位光电*) OR GVL_IO.I_Temp[6,7](*取UC站到位光电*) OR GVL_IO.I_Temp[6,8](*下工装站到位光电*) OR GVL_IO.I_Temp[6,10](*下UC皮带到位光电*) OR GVL_IO.I_Temp[6,12](*下工装皮带到位光电*)) ;
_arrFbErrorTag3[_i].Language[E_Language.Chinese]:="机台中有残余物料，请手动清料";
_arrFbErrorTag3[_i].Language[E_Language.English]:="There is a residue in the machine. Please clean the material manually";

_i:=1;
_arrFbErrorTag3[_i].ErrorTime:=T#5S;
_arrFbErrorTag3[_i].Enable:=GVL.stOverTime.bAcquireCheck2 AND GVL_P.G_stSystem.stMode.bAutoRunning;
_arrFbErrorTag3[_i].Language[E_Language.Chinese]:="接驳线光电检测超时";
_arrFbErrorTag3[_i].Language[E_Language.English]:="Relay line photoelectric detection timeout";

_i:=2;
_arrFbErrorTag3[_i].ErrorTime:=T#20S;
_arrFbErrorTag3[_i].Enable:=GVL.stOverTime.bLine0Check3 AND GVL_P.G_stSystem.stMode.bAutoRunning;
_arrFbErrorTag3[_i].Language[E_Language.Chinese]:="主流线到位光电检测超时";
_arrFbErrorTag3[_i].Language[E_Language.English]:="The mainstream line is in place to photoelectric test timeout";

_i:=3;
_arrFbErrorTag3[_i].ErrorTime:=T#5S;
_arrFbErrorTag3[_i].Enable:=GVL.stOverTime.bLine0Check2 AND GVL_P.G_stSystem.stMode.bAutoRunning;
_arrFbErrorTag3[_i].Language[E_Language.Chinese]:="主流线阻挡光电检测超时";
_arrFbErrorTag3[_i].Language[E_Language.English]:="The main line blocks the photoelectric detection timeout";

_i:=4;
_arrFbErrorTag3[_i].ErrorTime:=T#5S;
_arrFbErrorTag3[_i].Enable:=GVL.stOverTime.bUnloadFrockConveyorCheck2 AND GVL_P.G_stSystem.stMode.bAutoRunning;
_arrFbErrorTag3[_i].Language[E_Language.Chinese]:="下工装皮带到位光电检测超时";
_arrFbErrorTag3[_i].Language[E_Language.English]:="The next working belt is in the photoelectric detection timeout";

_i:=5;
_arrFbErrorTag3[_i].ErrorTime:=T#5S;
_arrFbErrorTag3[_i].Enable:=GVL.stOverTime.bUnloadUcCheck2 AND GVL_P.G_stSystem.stMode.bAutoRunning;
_arrFbErrorTag3[_i].Language[E_Language.Chinese]:="下UC皮带到位光电检测超时";
_arrFbErrorTag3[_i].Language[E_Language.English]:="The lower uc belt is in place to photoelectric test timeout";

_i:=6;
_arrFbErrorTag3[_i].ErrorTime:=T#5S;
_arrFbErrorTag3[_i].Enable:=NOT P_StationSteering._bManual AND GVL.stOverTime.bOpenLockCheck AND GVL_P.G_stSystem.stMode.bAutoRunning;
_arrFbErrorTag3[_i].Language[E_Language.Chinese]:="解锁站到位光电检测超时";
_arrFbErrorTag3[_i].Language[E_Language.English]:="The solution lock station is in place for photoelectric detection timeout";

_i:=7;
_arrFbErrorTag3[_i].ErrorTime:=T#5S;
_arrFbErrorTag3[_i].Enable:=GVL.stOverTime.bSteeringCheck1 AND GVL_P.G_stSystem.stMode.bAutoRunning;
_arrFbErrorTag3[_i].Language[E_Language.Chinese]:="转向站到位光电检测超时";
_arrFbErrorTag3[_i].Language[E_Language.English]:="Turn to the station to photoelectric test timeout";

_i:=8;
_arrFbErrorTag3[_i].ErrorTime:=T#5S;
_arrFbErrorTag3[_i].Enable:=GVL.stOverTime.bTakeUcCheck1 AND GVL_P.G_stSystem.stMode.bAutoRunning;
_arrFbErrorTag3[_i].Language[E_Language.Chinese]:="取UC站到位光电检测超时";
_arrFbErrorTag3[_i].Language[E_Language.English]:="The uc station is in place for photoelectric detection timeout";

_i:=9;
_arrFbErrorTag3[_i].ErrorTime:=T#5S;
_arrFbErrorTag3[_i].Enable:=GVL.stOverTime.bUnloadUcCheck1 AND GVL_P.G_stSystem.stMode.bAutoRunning;
_arrFbErrorTag3[_i].Language[E_Language.Chinese]:="翻转气缸到位光电检测超时";
_arrFbErrorTag3[_i].Language[E_Language.English]:="The inverted cylinder is in place for photoelectric detection timeout";

_i:=10;
_arrFbErrorTag3[_i].ErrorTime:=T#5S;
_arrFbErrorTag3[_i].Enable:=GVL.stOverTime.bUnloadFrockCheck1 AND GVL_P.G_stSystem.stMode.bAutoRunning;
_arrFbErrorTag3[_i].Language[E_Language.Chinese]:="下工装站到位光电检测超时";
_arrFbErrorTag3[_i].Language[E_Language.English]:="The next working station is in place for photoelectric detection timeout";

_i:=11;
_arrFbErrorTag3[_i].ErrorTime:=T#5S;
_arrFbErrorTag3[_i].Enable:=G_arrStation[E_Station.OpenLock].iStepNow=1100 AND GVL.I.bLine0Check1 AND NOT GVL.I.bLine0Check2 AND GVL_P.G_stSystem.stMode.bAutoRunning;
_arrFbErrorTag3[_i].Language[E_Language.Chinese]:="IN61 主流线阻挡光电检测超时";
_arrFbErrorTag3[_i].Language[E_Language.English]:="The IN61 Line0Check2 detection timeout";

_i:=12;
_arrFbErrorTag3[_i].ErrorTime:=T#0S;
_arrFbErrorTag3[_i].Enable:=GVL.stOverTime.bLine0PushElevatorUp AND GVL_P.G_stSystem.stMode.bAutoRunning;
_arrFbErrorTag3[_i].Language[E_Language.Chinese]:="拨料升降气缸上升速度过慢报警";
_arrFbErrorTag3[_i].Language[E_Language.English]:="The IN61 Line0Check2 detection timeout";

_i:=13;
_arrFbErrorTag3[_i].ErrorTime:=T#0S;
_arrFbErrorTag3[_i].Enable:=NOT GVL.I.bDoor AND GVL_P.G_stSystem.stMode.bAutoRunning AND NOT GVL.stSetting.bSafeDoorShield;
_arrFbErrorTag3[_i].Language[E_Language.Chinese]:="设备运行中安全门被打开";
_arrFbErrorTag3[_i].Language[E_Language.English]:="Safe door open in running";


(*_i:=10;
_arrFbErrorTag3[_i].Enable:=NOT GVL.I.bDoor;
_arrFbErrorTag3[_i].Language[E_Language.Chinese]:="安全门打开";*)

IF gvl_p.G_stSystem.stInput.bResetAlarm THEN
	GVL.stOverTime.bAcquireCheck2:=FALSE;
	GVL.stOverTime.bLine0Check2:=FALSE;
	GVL.stOverTime.bOpenLockCheck:=FALSE;
	GVL.stOverTime.bSteeringCheck1:=FALSE;
	GVL.stOverTime.bTakeUcCheck1:=FALSE;
	GVL.stOverTime.bUnloadFrockCheck1:=FALSE;
	GVL.stOverTime.bUnloadFrockConveyorCheck2:=FALSE;
	GVL.stOverTime.bUnloadUcCheck1:=FALSE;
	GVL.stOverTime.bUnloadUcCheck2:=FALSE;
	IF GVL.stOverTime.bLine0PushElevatorUp THEN
		GVL.stOverTime.bLine0PushElevatorUp:=FALSE;
		GVL.AlarmResetMark:=TRUE;
	END_IF
END_IF

FOR _i:=0 TO 20 BY 1 DO
_arrFbErrorTag3[_i](
	System:=G_stSystem , 
	Error:=G_stError , 
	ID:=TO_BYTE(53) , 
	Category:=E_ErrorCategory.Other , 
	InfoIndex:=TO_BYTE(_i) , 
	Enable:= , 
	Message:= , 
	Level:=3 , 
	Position:="P_Alarm:A_Alarm3" , 
	ErrorTime:= , 
	Language:= , 
	Erroring=> , 
	ErrorCode=> );
END_FOR
END_ACTION

ACTION A_Alarm4:








FOR _i:=0 TO 20 BY 1 DO
_arrFbErrorTag4[_i](
	System:=G_stSystem , 
	Error:=G_stError , 
	ID:=TO_BYTE(54) , 
	Category:=E_ErrorCategory.Other , 
	InfoIndex:=TO_BYTE(_i) , 
	Enable:= , 
	Message:= , 
	Level:=4 , 
	Position:="P_Alarm:A_Alarm4" , 
	ErrorTime:= , 
	Language:= , 
	Erroring=> , 
	ErrorCode=> );
END_FOR
END_ACTION

ACTION A_Alarm5:
_i:=0;
_arrFbErrorTag5[_i].Enable:=(G_stSystem.stMode.bHomeDone AND G_arrStation[E_Station.OpenLock].iStepNow = 1000) ;
_arrFbErrorTag5[_i].Language[E_Language.Chinese]:="请确认机台是否有残余物料,点击启动继续流程";
_arrFbErrorTag5[_i].Language[E_Language.English]:="Please confirm whether there is any residual material . Click the start continue process";

//_i:=1;
//_arrFbErrorTag5[_i].ErrorTime:=T#5S;
//_arrFbErrorTag5[_i].Enable:=NOT P_StationSteering._bManual AND GVL.stOverTime.bOpenLockCheck;
//_arrFbErrorTag5[_i].Language[E_Language.Chinese]:="解锁站到位光电检测超时";
//_arrFbErrorTag5[_i].Language[E_Language.English]:="The solution lock station is in place for photoelectric detection timeout";

//_i:=2;
//_arrFbErrorTag5[_i].ErrorTime:=T#5S;
//_arrFbErrorTag5[_i].Enable:=GVL.stOverTime.bSteeringCheck1;
//_arrFbErrorTag5[_i].Language[E_Language.Chinese]:="转向站到位光电检测超时";
//_arrFbErrorTag5[_i].Language[E_Language.English]:="Turn to the station to photoelectric test timeout";

//_i:=3;
//_arrFbErrorTag5[_i].ErrorTime:=T#5S;
//_arrFbErrorTag5[_i].Enable:=GVL.stOverTime.bTakeUcCheck1;
//_arrFbErrorTag5[_i].Language[E_Language.Chinese]:="取UC站到位光电检测超时";
//_arrFbErrorTag5[_i].Language[E_Language.English]:="The uc station is in place for photoelectric detection timeout";

//_i:=4;
//_arrFbErrorTag5[_i].ErrorTime:=T#5S;
//_arrFbErrorTag5[_i].Enable:=GVL.stOverTime.bUnloadUcCheck1;
//_arrFbErrorTag5[_i].Language[E_Language.Chinese]:="翻转气缸到位光电检测超时";
//_arrFbErrorTag5[_i].Language[E_Language.English]:="The inverted cylinder is in place for photoelectric detection timeout";

//_i:=5;
//_arrFbErrorTag5[_i].ErrorTime:=T#5S;
//_arrFbErrorTag5[_i].Enable:=GVL.stOverTime.bUnloadFrockCheck1;
//_arrFbErrorTag5[_i].Language[E_Language.Chinese]:="下工装站到位光电检测超时";
//_arrFbErrorTag5[_i].Language[E_Language.English]:="The next working station is in place for photoelectric detection timeout";



FOR _i:=0 TO 20 BY 1 DO
_arrFbErrorTag5[_i](
	System:=G_stSystem , 
	Error:=G_stError , 
	ID:=TO_BYTE(55) , 
	Category:=E_ErrorCategory.Other , 
	InfoIndex:=TO_BYTE(_i) , 
	Enable:= , 
	Message:= , 
	Level:=5 , 
	Position:="P_Alarm:A_Alarm5" , 
	ErrorTime:= , 
	Language:= , 
	Erroring=> , 
	ErrorCode=> );
END_FOR
END_ACTION

END_PROGRAM

// ---- POUs/P_StationSteering.TcPOU
PROGRAM P_StationSteering
VAR
	_station:					REFERENCE TO ST_SystemStation;
	
	_arrTemp:					ARRAY[0..10] OF BOOL;
	_bEnable: 					BOOL;
	
	_bManual:                   BOOL;//  手动上料

END_VAR

_station REF= G_arrStation[E_Station.Steering];
_station.arrName[E_Language.Chinese]:="转向站";
_station.arrName[E_Language.Vietnamese]:="Quay về vị trí";
_bEnable:=NOT GVL.stSetting.arrStationShield[E_Station.Steering];
A_Home();
A_Auto();

_bManual:=GVL.stSetting.bManualLoad ;

ACTION A_Auto:
CASE _station.iStepNow OF
	1000:
		_station.arrInfo[E_Language.Chinese]:="初始化完成等待启动";
		IF  _bEnable THEN
			_station.iStepNext:=1101;
		END_IF
	1101:
		_station.arrInfo[E_Language.Chinese]:="判断是否有料";
		IF NOT GVL.I.bSteeringCheck1 THEN
			_station.iStepNext:=SEL(_bManual,1201,1551);
		END_IF
	1201:
		_station.arrInfo[E_Language.Chinese]:="请求放料";
		GVL.stHandshake.bSteering:=TRUE;
		IF GVL.stHandshake.bSteeringOk THEN
			_station.iStepNext:=1301;
		END_IF
	1301:
	     _station.arrInfo[E_Language.Chinese]:="检测物料是否到转向站";
		 GVL.stOverTime.bSteeringCheck1:=TRUE;
	    IF GVL.I.bSteeringCheck1 THEN
			GVL.stOverTime.bSteeringCheck1:=FALSE;
			_station.iStepNext:=1311;
		END_IF
	1311:
		_station.arrInfo[E_Language.Chinese]:="复位放料请求";
		GVL.stHandshake.bSteering:=FALSE;
		IF NOT  GVL.stHandshake.bSteeringOk THEN
			_station.iStepNext:=1351;
		END_IF
	1351:
		_station.arrInfo[E_Language.Chinese]:="限位气缸缩回";
		IF  G_arrFbCylinder[E_Cylinder.SteeringAcquireLimit].M_HomeRequest() THEN
			_station.iStepNext:=1401;
		END_IF
	1401:
		_station.arrInfo[E_Language.Chinese]:="顶升气缸伸出";
		IF M_LiftWork() THEN
			_station.iStepNext:=1451;
	    END_IF
	1451:
		_station.arrInfo[E_Language.Chinese]:="接驳升降气缸缩回";
		CASE GVL_Data.stRecipe.eMachineType OF
			E_MachineType._367:
				IF  G_arrFbCylinder[E_Cylinder.SteeringAcquireElevator].M_HomeRequest() THEN
					_station.iStepNext:=1501;
		    	END_IF
			ELSE
				_station.iStepNext:=1501;
		END_CASE
	1501:
		_station.arrInfo[E_Language.Chinese]:="旋转气缸动作";
		IF M_RotateWork() THEN
			_station.iStepNext:=1551;
		END_IF
	1551:
		_station.arrInfo[E_Language.Chinese]:="等待解锁站请求放料";
		IF GVL.stHandshake.bOpenToSteering THEN
			GVL.stHandshake.bSteeringToOpen:=TRUE;
			_station.iStepNext:=SEL(_bManual,1561,1651);
		END_IF
	1561:
		_station.arrInfo[E_Language.Chinese]:="接驳升降气缸缩回";
        IF  G_arrFbCylinder[E_Cylinder.SteeringAcquireElevator].M_HomeRequest() THEN
			_station.iStepNext:=1601;
		END_IF
	1601:
		_station.arrInfo[E_Language.Chinese]:="顶升气缸缩回";
		IF M_LiftHome() THEN
			_station.iStepNext:=1651;
		END_IF
	1651:
		_station.arrInfo[E_Language.Chinese]:="等待复位放料请求";
		IF NOT GVL.stHandshake.bOpenToSteering THEN
			GVL.stHandshake.bSteeringToOpen:=FALSE;
			_station.iStepNext:=SEL(_bManual,1655,1101);
		END_IF
	1655:
		CASE GVL_Data.stRecipe.eMachineType OF
			E_MachineType._311:
				_station.iStepNext:=1661;
			E_MachineType._367:	
				GVL.stHandshake.bSteering:=TRUE;
				_station.iStepNext:=1701;		
			ELSE
				_station.iStepNext:=1701;
		END_CASE
	1661:
		_station.arrInfo[E_Language.Chinese]:="顶升气缸伸出";
		IF M_LiftWork() THEN
			_station.iStepNext:=1671;
		END_IF
	1671:
		_station.arrInfo[E_Language.Chinese]:="旋转气缸复位";
		IF M_RotateHome() THEN
			_station.iStepNext:=1681;
		END_IF
	1681:
		_station.arrInfo[E_Language.Chinese]:="顶升气缸缩回";
		IF M_LiftHome() THEN
			_station.iStepNext:=1701;
		END_IF
	1701:
		_station.arrInfo[E_Language.Chinese]:="接驳升降气缸伸出 限位气缸伸出";
		IF G_arrFbCylinder[E_Cylinder.SteeringAcquireElevator].M_WorkRequest() and G_arrFbCylinder[E_Cylinder.SteeringAcquireLimit].M_WorkRequest() THEN
			_station.iStepNext:=1901;
		END_IF
	1901:
		_station.arrInfo[E_Language.Chinese]:="旋转气缸复位"; 
		IF M_RotateHome() THEN
			_station.iStepNext:=SEL(GVL_Data.stRecipe.eMachineType=E_MachineType._367,1101,1201);
		END_IF
END_CASE
END_ACTION

ACTION A_Home:
CASE _station.iStepNow OF
	0:
		_station.arrInfo[E_Language.Chinese]:="等待初始化";
		_station.iStepNext:=SEL(_bEnable,1000,100);
	100:
	    IF GVL_Data.stRecipe.eMachineType = E_MachineType._367 THEN
			_station.iStepNext:=150;
			ELSE
				_station.iStepNext:=450;
		END_IF
	150:
		_station.arrInfo[E_Language.Chinese]:="顶升气缸伸出";
		    IF G_arrFbCylinder[E_Cylinder.SteeringLift].M_WorkRequest() THEN
		     	_station.iStepNext:=200;
		    END_IF
		
	200:
		_station.arrInfo[E_Language.Chinese]:="接驳升降气缸缩回";
		IF G_arrFbCylinder[E_Cylinder.SteeringAcquireElevator].M_HomeRequest()  THEN
			_station.iStepNext:=300;
		END_IF
	
	300:
		_station.arrInfo[E_Language.Chinese]:="旋转气缸复位";
		IF G_arrFbCylinder[E_Cylinder.SteeringRotate].M_HomeRequest() THEN
			_station.iStepNext:=400;
		END_IF
	400:
		_station.arrInfo[E_Language.Chinese]:="顶升气缸缩回";
		IF G_arrFbCylinder[E_Cylinder.SteeringLift].M_HomeRequest() THEN
			_station.iStepNext:=450;
		END_IF
	450:
		IF NOT _bManual THEN
			_station.iStepNext:=500;
		ELSE
			_station.iStepNext:=700;
		END_IF
	500:
		_station.arrInfo[E_Language.Chinese]:="接驳升降气缸伸出";
		IF G_arrFbCylinder[E_Cylinder.SteeringAcquireElevator].M_WorkRequest()  THEN
			_station.iStepNext:=600;
		END_IF
	600:
		_station.arrInfo[E_Language.Chinese]:="限位气缸伸出";
		IF  G_arrFbCylinder[E_Cylinder.SteeringAcquireLimit].M_WorkRequest() THEN
			_station.iStepNext:=1000;
		END_IF
		
		
	700:
	    _station.arrInfo[E_Language.Chinese]:="接驳升降气缸缩回";
		IF G_arrFbCylinder[E_Cylinder.SteeringAcquireElevator].M_HomeRequest()  THEN
			_station.iStepNext:=800;
		END_IF
	800:
	    _station.arrInfo[E_Language.Chinese]:="限位气缸缩回";
		IF  G_arrFbCylinder[E_Cylinder.SteeringAcquireLimit].M_HomeRequest() THEN
			_station.iStepNext:=1000;
		END_IF
		
	
END_CASE
END_ACTION

METHOD M_LiftHome : BOOL
VAR_INPUT
END_VAR
CASE GVL_Data.stRecipe.eMachineType OF
	E_MachineType._367:
		M_LiftHome:=G_arrFbCylinder[E_Cylinder.SteeringLift].M_HomeRequest();
	ELSE
		M_LiftHome:=TRUE;		
END_CASE
END_METHOD

METHOD M_LiftWork : BOOL
VAR_INPUT
END_VAR
CASE GVL_Data.stRecipe.eMachineType OF
	E_MachineType._367:	
		M_LiftWork:=G_arrFbCylinder[E_Cylinder.SteeringLift].M_WorkRequest();
	ELSE
		M_LiftWork:=TRUE;
END_CASE
END_METHOD

METHOD M_RotateHome : BOOL
VAR_INPUT
END_VAR
CASE GVL_Data.stRecipe.eMachineType OF
	E_MachineType._367:
		M_RotateHome:=G_arrFbCylinder[E_Cylinder.SteeringRotate].M_HomeRequest();
	ELSE
		M_RotateHome:=TRUE;	
END_CASE
END_METHOD

METHOD M_RotateWork : BOOL
VAR_INPUT
END_VAR
CASE GVL_Data.stRecipe.eMachineType OF
	E_MachineType._367:
		M_RotateWork:=G_arrFbCylinder[E_Cylinder.SteeringRotate].M_WorkRequest();
	ELSE
		M_RotateWork:=TRUE;
END_CASE
END_METHOD

END_PROGRAM

// ---- POUs/P_Device.TcPOU
PROGRAM P_Device
VAR
	_i:					INT;
	_t:					INT;
	_bFirstRun:			BOOL:=TRUE;
	_fbPulse:			FB_Pulse;
	_arrInput:			ARRAY[0..7,0..15] OF  BOOL;
	_arrOutput:			ARRAY[0..6,0..15] OF  BOOL;
	_arrTonInput :		ARRAY[0..7,0..15] OF  TON;
	_arrTonOutput:		ARRAY[0..6,0..15] OF  TON;
	_arrCylTon_H:		ARRAY[0..50] OF TON;
	_arrCylTon_W:		ARRAY[0..50] OF TON;
	
	
	_boolTemp:			POINTER TO BOOL;
	
	_eMachineType:		E_MachineType;
	_eMachineType1:		E_MachineType;

END_VAR

IF _bFirstRun THEN
	A_Info();
	_bFirstRun:=FALSE;
END_IF

A_InOut();// 输入输出
A_Axis();// 轴控制
A_Line();// 线体控制

IF GVL.stSetting.bDryRun THEN
	(*CASE GVL_Data.stRecipe.eMachineType OF
		E_MachineType._367:
	          A_CylinderTest367();
		E_MachineType._200:
		      A_CylinderTest201();
		E_MachineType._373:
		      A_CylinderTest373();
		E_MachineType._069:
		      A_CylinderTest069();
		E_MachineType._311:
		     A_CylinderTest311();
	END_CASE*)
	A_CylinderTest();
ELSE
	A_Cylinder();
END_IF

// 气缸屏蔽
IF GVL_Data.stRecipe.eMachineType<>_eMachineType1 THEN
	FOR _i:=0 TO 50 BY 1 DO
	G_arrCylinder[_i].stLock.bShield:=FALSE;
    END_FOR
	_eMachineType1:=GVL_Data.stRecipe.eMachineType;
END_IF


CASE GVL_Data.stRecipe.eMachineType OF
	E_MachineType._367:
		G_arrCylinder[E_Cylinder.AcquirePrevent0].stLock.bShield:=TRUE;
		G_arrCylinder[E_Cylinder.AcquirePrevent1].stLock.bShield:=TRUE;
		G_arrCylinder[E_Cylinder.AcquireLift].stLock.bShield:=TRUE;
		G_arrCylinder[E_Cylinder.AcquirePush].stLock.bShield:=TRUE;
		G_arrCylinder[E_Cylinder.AcquireElevator].stLock.bShield:=TRUE;
		G_arrCylinder[E_Cylinder.UnloadFrockPrevent].stLock.bShield:=TRUE;
		G_arrCylinder[E_Cylinder.UnloadFrockLift].stLock.bShield:=TRUE;
		G_arrCylinder[E_Cylinder.UnloadUcBeltTipper].stLock.bShield:=TRUE;
		G_arrCylinder[E_Cylinder.UnloadUcBeltLift].stLock.bShield:=TRUE;
		G_arrCylinder[E_Cylinder.OpenLockElevator].stLock.bShield:=TRUE;
		G_arrCylinder[E_Cylinder.OpenLockPin].stLock.bShield:=TRUE;
		G_arrCylinder[E_Cylinder.TakeUcElevator].stLock.bShield:=TRUE;
		G_arrCylinder[E_Cylinder.TakeUcPush1].stLock.bShield:=TRUE;
		G_arrCylinder[E_Cylinder.OpenLockTranslation].stLock.bShield:=TRUE;
		G_arrCylinder[E_Cylinder.OpenLockPressPush].stLock.bShield:=TRUE;
		G_arrCylinder[E_Cylinder.OpenLockPressRotate].stLock.bShield:=TRUE;
		G_arrCylinder[E_Cylinder.AcquirePrevent2].stLock.bShield:=TRUE;
		
	E_MachineType._200:
		G_arrCylinder[E_Cylinder.TakeUcStandard].stLock.bShield:=TRUE;
		G_arrCylinder[E_Cylinder.OpenLockElevator].stLock.bShield:=TRUE;
		G_arrCylinder[E_Cylinder.OpenLockPin].stLock.bShield:=TRUE;
		G_arrCylinder[E_Cylinder.TakeUcElevator].stLock.bShield:=TRUE;
		G_arrCylinder[E_Cylinder.TakeUcPush1].stLock.bShield:=TRUE;
		G_arrCylinder[E_Cylinder.OpenLockTranslation].stLock.bShield:=TRUE;
		G_arrCylinder[E_Cylinder.TakeUcFrockClamp].stLock.bShield:=TRUE;
		G_arrCylinder[E_Cylinder.OpenLockPressPush].stLock.bShield:=TRUE;
		G_arrCylinder[E_Cylinder.OpenLockPressRotate].stLock.bShield:=TRUE;
		G_arrCylinder[E_Cylinder.SteeringLift].stLock.bShield:=TRUE;
		G_arrCylinder[E_Cylinder.SteeringRotate].stLock.bShield:=TRUE;
		G_arrCylinder[E_Cylinder.Line0PushElevator].stLock.bShield:=TRUE;
	E_MachineType._373:
		G_arrCylinder[E_Cylinder.OpenLockPush2].stLock.bShield:=TRUE;
		G_arrCylinder[E_Cylinder.UnloadFrockLift].stLock.bShield:=TRUE;
		G_arrCylinder[E_Cylinder.UnloadFrockPrevent].stLock.bShield:=TRUE;
		G_arrCylinder[E_Cylinder.UnloadUcBeltTipper].stLock.bShield:=TRUE;
		G_arrCylinder[E_Cylinder.UnloadUcBeltLift].stLock.bShield:=TRUE;
		G_arrCylinder[E_Cylinder.OpenLockElevator].stLock.bShield:=TRUE;
		G_arrCylinder[E_Cylinder.OpenLockPin].stLock.bShield:=TRUE;
		G_arrCylinder[E_Cylinder.TakeUcElevator].stLock.bShield:=TRUE;
		G_arrCylinder[E_Cylinder.TakeUcPush1].stLock.bShield:=TRUE;
		G_arrCylinder[E_Cylinder.OpenLockTranslation].stLock.bShield:=TRUE;
		G_arrCylinder[E_Cylinder.TakeUc1Z2].stLock.bShield:=TRUE;
		G_arrCylinder[E_Cylinder.TakeUcFrockClamp].stLock.bShield:=TRUE;
		G_arrCylinder[E_Cylinder.TakeUcStandard].stLock.bShield:=TRUE;
		G_arrCylinder[E_Cylinder.SteeringLift].stLock.bShield:=TRUE;
		G_arrCylinder[E_Cylinder.SteeringRotate].stLock.bShield:=TRUE;
		G_arrCylinder[E_Cylinder.Line0PushElevator].stLock.bShield:=TRUE;
	E_MachineType._069:
		G_arrCylinder[E_Cylinder.TakeUcStandard].stLock.bShield:=TRUE;
		G_arrCylinder[E_Cylinder.UnloadFrockPrevent].stLock.bShield:=TRUE;
		G_arrCylinder[E_Cylinder.UnloadFrockLift].stLock.bShield:=TRUE;
		G_arrCylinder[E_Cylinder.UnloadUcBeltTipper].stLock.bShield:=TRUE;
		G_arrCylinder[E_Cylinder.UnloadUcBeltLift].stLock.bShield:=TRUE;
		G_arrCylinder[E_Cylinder.OpenLockElevator].stLock.bShield:=TRUE;
		G_arrCylinder[E_Cylinder.OpenLockPin].stLock.bShield:=TRUE;
		G_arrCylinder[E_Cylinder.TakeUcElevator].stLock.bShield:=TRUE;
		G_arrCylinder[E_Cylinder.TakeUcPush1].stLock.bShield:=TRUE;
		G_arrCylinder[E_Cylinder.OpenLockTranslation].stLock.bShield:=TRUE;
		G_arrCylinder[E_Cylinder.TakeUcFrockClamp].stLock.bShield:=TRUE;
		G_arrCylinder[E_Cylinder.OpenLockPressPush].stLock.bShield:=TRUE;
		G_arrCylinder[E_Cylinder.OpenLockPressRotate].stLock.bShield:=TRUE;
		G_arrCylinder[E_Cylinder.SteeringLift].stLock.bShield:=TRUE;
		G_arrCylinder[E_Cylinder.SteeringRotate].stLock.bShield:=TRUE;
		G_arrCylinder[E_Cylinder.Line0PushElevator].stLock.bShield:=TRUE;
	E_MachineType._311:
		G_arrCylinder[E_Cylinder.OpenLockPush].stLock.bShield:=TRUE;
		G_arrCylinder[E_Cylinder.OpenLockPush2].stLock.bShield:=TRUE;
		G_arrCylinder[E_Cylinder.TakeUcStandard].stLock.bShield:=TRUE;
		G_arrCylinder[E_Cylinder.UnloadFrockLift].stLock.bShield:=TRUE;
		G_arrCylinder[E_Cylinder.UnloadUcBeltTipper].stLock.bShield:=TRUE;
		G_arrCylinder[E_Cylinder.UnloadUcBeltLift].stLock.bShield:=TRUE;
		G_arrCylinder[E_Cylinder.UnloadFrockPrevent].stLock.bShield:=TRUE;
		G_arrCylinder[E_Cylinder.TakeUcFrockClamp].stLock.bShield:=TRUE;
		G_arrCylinder[E_Cylinder.OpenLockPressPush].stLock.bShield:=TRUE;
		G_arrCylinder[E_Cylinder.OpenLockPressRotate].stLock.bShield:=TRUE;
		G_arrCylinder[E_Cylinder.SteeringLift].stLock.bShield:=TRUE;
		G_arrCylinder[E_Cylinder.SteeringRotate].stLock.bShield:=TRUE;
		G_arrCylinder[E_Cylinder.Line0PushElevator].stLock.bShield:=TRUE;

		
END_CASE

ACTION A_Axis:
_i:=E_Axis.Z;
G_arrAxis[_i].arrInfo[E_Language.Chinese].sName:="Z轴";
G_arrAxis[_i].arrInfo[E_Language.English].sName:="Z";
G_arrAxis[_i].arrInfo[E_Language.Vietnamese].sName:="Z";
G_arrAxis[_i].stLock.bShield:=GVL_Data.stRecipe.eMachineType=E_MachineType._200;
G_arrAxis[_i].stInput.bNegative:=GVL_IO.AxisInput.0;
G_arrAxis[_i].stInput.bPositive:=GVL_IO.AxisInput.2;
G_arrAxisData[_i].stMode.iHomeMode:=0;
END_ACTION

ACTION A_Cylinder:
_i:=E_Cylinder.Line0Part;
G_arrCylinder[_i].stInput.bHome:=GVL.I.bLine0Part_Cyl_H;
G_arrCylinder[_i].stInput.bWork:=GVL.I.bLine0Part_Cyl_W;
GVL.Q.bLine0Part_Cyl_H:=G_arrCylinder[_i].stOutput.bHome;
GVL.Q.bLine0Part_Cyl_W:=G_arrCylinder[_i].stOutput.bWork;

_i:=E_Cylinder.Line0Prevent;
G_arrCylinder[_i].stInput.bHome:=GVL.I.bLine0Prevent_Cyl_H;
G_arrCylinder[_i].stInput.bWork:=GVL.I.bLine0Prevent_Cyl_W;
GVL.Q.bLine0Prevent_Cyl_H:=G_arrCylinder[_i].stOutput.bHome;
GVL.Q.bLine0Prevent_Cyl_W:=G_arrCylinder[_i].stOutput.bWork;

_i:=E_Cylinder.Line0Push;
G_arrCylinder[_i].stInput.bHome:=GVL.I.bLine0Push_Cyl_H;
G_arrCylinder[_i].stInput.bWork:=GVL.I.bLine0Push_Cyl_W;
GVL.Q.bLine0Push_Cyl_H:=G_arrCylinder[_i].stOutput.bHome;
GVL.Q.bLine0Push_Cyl_W:=G_arrCylinder[_i].stOutput.bWork;

_i:=E_Cylinder.AcquirePrevent0;
G_arrCylinder[_i].stInput.bHome:=NOT GVL.I.bAcquirePrevent0_Cyl_W;
G_arrCylinder[_i].stInput.bWork:=GVL.I.bAcquirePrevent0_Cyl_W;
GVL.Q.bAcquirePrevent0_Cyl_H:=G_arrCylinder[_i].stOutput.bHome;
GVL.Q.bAcquirePrevent0_Cyl_W:=G_arrCylinder[_i].stOutput.bWork;

_i:=E_Cylinder.AcquirePrevent1;
G_arrCylinder[_i].stInput.bHome:=NOT GVL.I.bAcquirePrevent1_Cyl_W;
G_arrCylinder[_i].stInput.bWork:=GVL.I.bAcquirePrevent1_Cyl_W;
GVL.Q.bAcquirePrevent1_Cyl_H:=G_arrCylinder[_i].stOutput.bHome;
GVL.Q.bAcquirePrevent1_Cyl_W:=G_arrCylinder[_i].stOutput.bWork;

_i:=E_Cylinder.AcquireLift;
G_arrCylinder[_i].stInput.bHome:=GVL.I.bAcquireLift_Cyl_H;
G_arrCylinder[_i].stInput.bWork:=GVL.I.bAcquireLift_Cyl_W;
GVL.Q.bAcquireLift_Cyl_H:=G_arrCylinder[_i].stOutput.bHome;
GVL.Q.bAcquireLift_Cyl_W:=G_arrCylinder[_i].stOutput.bWork;

_i:=E_Cylinder.AcquirePush;
G_arrCylinder[_i].stInput.bHome:=GVL.I.bAcquirePush_Cyl_H;
G_arrCylinder[_i].stInput.bWork:=GVL.I.bAcquirePush_Cyl_W;
GVL.Q.bAcquirePush_Cyl_H:=G_arrCylinder[_i].stOutput.bHome;
GVL.Q.bAcquirePush_Cyl_W:=G_arrCylinder[_i].stOutput.bWork;

_i:=E_Cylinder.AcquireElevator;
G_arrCylinder[_i].stInput.bHome:=GVL.I.bAcquireElevator_Cyl_H;
G_arrCylinder[_i].stInput.bWork:=GVL.I.bAcquireElevator_Cyl_W;
GVL.Q.bAcquireElevator_Cyl_H:=G_arrCylinder[_i].stOutput.bHome;
GVL.Q.bAcquireElevator_Cyl_W:=G_arrCylinder[_i].stOutput.bWork;

_i:=E_Cylinder.SteeringLift;
G_arrCylinder[_i].stInput.bHome:=GVL.I.bSteeringLift_Cyl_H;
G_arrCylinder[_i].stInput.bWork:=GVL.I.bSteeringLift_Cyl_W;
GVL.Q.bSteeringLift_Cyl_H:=G_arrCylinder[_i].stOutput.bHome;
GVL.Q.bSteeringLift_Cyl_W:=G_arrCylinder[_i].stOutput.bWork;

_i:=E_Cylinder.SteeringAcquireElevator;
G_arrCylinder[_i].stInput.bHome:=GVL.I.bSteeringAcquireElevator_Cyl_H;
G_arrCylinder[_i].stInput.bWork:=GVL.I.bSteeringAcquireElevator_Cyl_W;
GVL.Q.bSteeringAcquireElevator_Cyl_H:=G_arrCylinder[_i].stOutput.bHome;
GVL.Q.bSteeringAcquireElevator_Cyl_W:=G_arrCylinder[_i].stOutput.bWork;

_i:=E_Cylinder.SteeringRotate;
G_arrCylinder[_i].stInput.bHome:=GVL.I.bSteeringRotate_Cyl_H;
G_arrCylinder[_i].stInput.bWork:=GVL.I.bSteeringRotate_Cyl_W;
GVL.Q.bSteeringRotate_Cyl_H:=G_arrCylinder[_i].stOutput.bHome;
GVL.Q.bSteeringRotate_Cyl_W:=G_arrCylinder[_i].stOutput.bWork;

_i:=E_Cylinder.SteeringAcquireLimit;
G_arrCylinder[_i].stInput.bHome:=GVL.I.bSteeringAcquireLimit_Cyl_H;
G_arrCylinder[_i].stInput.bWork:=GVL.I.bSteeringAcquireLimit_Cyl_W;
GVL.Q.bSteeringAcquireLimit_Cyl_H:=G_arrCylinder[_i].stOutput.bHome;
GVL.Q.bSteeringAcquireLimit_Cyl_W:=G_arrCylinder[_i].stOutput.bWork;

_i:=E_Cylinder.OpenLockPrevent;
G_arrCylinder[_i].stInput.bHome:=NOT GVL.I.bOpenLockPrevent_Cyl_W;
G_arrCylinder[_i].stInput.bWork:=GVL.I.bOpenLockPrevent_Cyl_W;
GVL.Q.bOpenLockPrevent_Cyl_H:=G_arrCylinder[_i].stOutput.bHome;
GVL.Q.bOpenLockPrevent_Cyl_W:=G_arrCylinder[_i].stOutput.bWork;

_i:=E_Cylinder.OpenLockLift;
G_arrCylinder[_i].stInput.bHome:=GVL.I.bOpenLockLift_Cyl_H;
G_arrCylinder[_i].stInput.bWork:=GVL.I.bOpenLockLift_Cyl_W;
GVL.Q.bOpenLockLift_Cyl_H:=G_arrCylinder[_i].stOutput.bHome;
GVL.Q.bOpenLockLift_Cyl_W:=G_arrCylinder[_i].stOutput.bWork;

_i:=E_Cylinder.OpenLockPush;
G_arrCylinder[_i].stInput.bHome:=GVL.I.bOpenLockPush_Cyl_H;
G_arrCylinder[_i].stInput.bWork:=GVL.I.bOpenLockPush_Cyl_W;
GVL.Q.bOpenLockPush_Cyl_H:=G_arrCylinder[_i].stOutput.bHome;
GVL.Q.bOpenLockPush_Cyl_W:=G_arrCylinder[_i].stOutput.bWork;

_i:=E_Cylinder.OpenLockRotate;
G_arrCylinder[_i].stInput.bHome:=GVL.I.bOpenLockRotate_Cyl_H;
G_arrCylinder[_i].stInput.bWork:=GVL.I.bOpenLockRotate_Cyl_W;
GVL.Q.bOpenLockRotate_Cyl_H:=G_arrCylinder[_i].stOutput.bHome;
GVL.Q.bOpenLockRotate_Cyl_W:=G_arrCylinder[_i].stOutput.bWork;

_i:=E_Cylinder.OpenLockPush2;
//G_arrCylinder[_i].stInput.bHome:=GVL.I.bOpenLockPush2_Cyl_H;
G_arrCylinder[_i].stInput.bHome:=NOT GVL.I.bOpenLockPush2_Cyl_W;
G_arrCylinder[_i].stInput.bWork:=GVL.I.bOpenLockPush2_Cyl_W;
GVL.Q.bOpenLockPush2_Cyl_H:=G_arrCylinder[_i].stOutput.bHome;
GVL.Q.bOpenLockPush2_Cyl_W:=G_arrCylinder[_i].stOutput.bWork;

_i:=E_Cylinder.TakeUcPrevent;
G_arrCylinder[_i].stInput.bHome:=NOT GVL.I.bTakeUcPrevent_Cyl_W;
G_arrCylinder[_i].stInput.bWork:=GVL.I.bTakeUcPrevent_Cyl_W;
GVL.Q.bTakeUcPrevent_Cyl_H:=G_arrCylinder[_i].stOutput.bHome;
GVL.Q.bTakeUcPrevent_Cyl_W:=G_arrCylinder[_i].stOutput.bWork;

_i:=E_Cylinder.TakeUcLift;
G_arrCylinder[_i].stInput.bHome:=GVL.I.bTakeUcLift_Cyl_H;
G_arrCylinder[_i].stInput.bWork:=GVL.I.bTakeUcLift_Cyl_W;
GVL.Q.bTakeUcLift_Cyl_H:=G_arrCylinder[_i].stOutput.bHome;
GVL.Q.bTakeUcLift_Cyl_W:=G_arrCylinder[_i].stOutput.bWork;

_i:=E_Cylinder.TakeUcPush;
G_arrCylinder[_i].stInput.bHome:=GVL.I.bTakeUcPush_Cyl_H;
G_arrCylinder[_i].stInput.bWork:=GVL.I.bTakeUcPush_Cyl_W;
GVL.Q.bTakeUcPush_Cyl_H:=G_arrCylinder[_i].stOutput.bHome;
GVL.Q.bTakeUcPush_Cyl_W:=G_arrCylinder[_i].stOutput.bWork;

_i:=E_Cylinder.TakeUcRotate;
G_arrCylinder[_i].stInput.bHome:=GVL.I.bTakeUcRotate_Cyl_H;
G_arrCylinder[_i].stInput.bWork:=GVL.I.bTakeUcRotate_Cyl_W;
GVL.Q.bTakeUcRotate_Cyl_H:=G_arrCylinder[_i].stOutput.bHome;
GVL.Q.bTakeUcRotate_Cyl_W:=G_arrCylinder[_i].stOutput.bWork;

_i:=E_Cylinder.TakeUcStandard;
G_arrCylinder[_i].stInput.bHome:=GVL.I.bTakeUcStandard_Cyl_H;
G_arrCylinder[_i].stInput.bWork:=GVL.I.bTakeUcStandard_Cyl_W;
GVL.Q.bTakeUcStandard_Cyl_H:=G_arrCylinder[_i].stOutput.bHome;
GVL.Q.bTakeUcStandard_Cyl_W:=G_arrCylinder[_i].stOutput.bWork;

_i:=E_Cylinder.UnloadFrockPrevent;
G_arrCylinder[_i].stInput.bHome:=NOT GVL.I.bUnloadFrockPrevent_Cyl_W;
G_arrCylinder[_i].stInput.bWork:=GVL.I.bUnloadFrockPrevent_Cyl_W;
GVL.Q.bUnloadFrockPrevent_Cyl_H:=G_arrCylinder[_i].stOutput.bHome;
GVL.Q.bUnloadFrockPrevent_Cyl_W:=G_arrCylinder[_i].stOutput.bWork;

_i:=E_Cylinder.UnloadFrockLift;
G_arrCylinder[_i].stInput.bHome:=GVL.I.bUnloadFrockLift_Cyl_H;
G_arrCylinder[_i].stInput.bWork:=GVL.I.bUnloadFrockLift_Cyl_W;
GVL.Q.bUnloadFrockLift_Cyl_H:=G_arrCylinder[_i].stOutput.bHome;
GVL.Q.bUnloadFrockLift_Cyl_W:=G_arrCylinder[_i].stOutput.bWork;

_i:=E_Cylinder.UnloadFrockPush;
G_arrCylinder[_i].stInput.bHome:=GVL.I.bUnloadFrockPush_Cyl_H;
G_arrCylinder[_i].stInput.bWork:=GVL.I.bUnloadFrockPush_Cyl_W;
GVL.Q.bUnloadFrockPush_Cyl_H:=G_arrCylinder[_i].stOutput.bHome;
GVL.Q.bUnloadFrockPush_Cyl_W:=G_arrCylinder[_i].stOutput.bWork;

_i:=E_Cylinder.TakeUc1Y;
G_arrCylinder[_i].stInput.bHome:=GVL.I.bTakeUc1Y_Cyl_H;
G_arrCylinder[_i].stInput.bWork:=GVL.I.bTakeUc1Y_Cyl_W;
GVL.Q.bTakeUc1Y_Cyl_H:=G_arrCylinder[_i].stOutput.bHome;
GVL.Q.bTakeUc1Y_Cyl_W:=G_arrCylinder[_i].stOutput.bWork;

_i:=E_Cylinder.TakeUc1Z1;
G_arrCylinder[_i].stInput.bHome:=GVL.I.bTakeUc1Z1_Cyl_H;
G_arrCylinder[_i].stInput.bWork:=GVL.I.bTakeUc1Z1_Cyl_W;
GVL.Q.bTakeUc1Z1_Cyl_H:=G_arrCylinder[_i].stOutput.bHome;
GVL.Q.bTakeUc1Z1_Cyl_W:=G_arrCylinder[_i].stOutput.bWork;

_i:=E_Cylinder.TakeUc1Z2;
G_arrCylinder[_i].stInput.bHome:=GVL.I.bTakeUc1Z2_Cyl_H;
G_arrCylinder[_i].stInput.bWork:=GVL.I.bTakeUc1Z2_Cyl_W;
GVL.Q.bTakeUc1Z2_Cyl_H:=G_arrCylinder[_i].stOutput.bHome;
GVL.Q.bTakeUc1Z2_Cyl_W:=G_arrCylinder[_i].stOutput.bWork;

_i:=E_Cylinder.TakeUc1Rotate;
G_arrCylinder[_i].stInput.bHome:=GVL.I.bTakeUc1Rotate_Cyl_H;
G_arrCylinder[_i].stInput.bWork:=GVL.I.bTakeUc1Rotate_Cyl_W;
GVL.Q.bTakeUc1Rotate_Cyl_H:=G_arrCylinder[_i].stOutput.bHome;
GVL.Q.bTakeUc1Rotate_Cyl_W:=G_arrCylinder[_i].stOutput.bWork;

_i:=E_Cylinder.TakeUc1Clamp;
G_arrCylinder[_i].stInput.bHome:=GVL.I.bTakeUc1Clamp_Cyl_H;
G_arrCylinder[_i].stInput.bWork:=GVL.I.bTakeUc1Clamp_Cyl_W;
GVL.Q.bTakeUc1Clamp_Cyl_H:=G_arrCylinder[_i].stOutput.bHome;
GVL.Q.bTakeUc1Clamp_Cyl_W:=G_arrCylinder[_i].stOutput.bWork;


_i:=E_Cylinder.UnloadUcElevator;
G_arrCylinder[_i].stInput.bHome:=GVL.I.bUnloadUcElevator_Cyl_H;
G_arrCylinder[_i].stInput.bWork:=GVL.I.bUnloadUcElevator_Cyl_W;
GVL.Q.bUnloadUcElevator_Cyl_H:=G_arrCylinder[_i].stOutput.bHome;
GVL.Q.bUnloadUcElevator_Cyl_W:=G_arrCylinder[_i].stOutput.bWork;


_i:=E_Cylinder.UnloadUcConveyorPush;
G_arrCylinder[_i].stInput.bHome:=GVL.I.bUnloadUcConveyorPush_Cyl_H;
G_arrCylinder[_i].stInput.bWork:=GVL.I.bUnloadUcConveyorPush_Cyl_W;
GVL.Q.bUnloadUcConveyorPush_Cyl_H:=G_arrCylinder[_i].stOutput.bHome;
GVL.Q.bUnloadUcConveyorPush_Cyl_W:=G_arrCylinder[_i].stOutput.bWork;


_i:=E_Cylinder.UnloadFrockConveyorPrevent;
G_arrCylinder[_i].stInput.bHome:=GVL.I.bUnloadFrockConveyorPrevent_Cyl_H;
G_arrCylinder[_i].stInput.bWork:=GVL.I.bUnloadFrockConveyorPrevent_Cyl_W;
GVL.Q.bUnloadFrockConveyorPrevent_Cyl_H:=G_arrCylinder[_i].stOutput.bHome;
GVL.Q.bUnloadFrockConveyorPrevent_Cyl_W:=G_arrCylinder[_i].stOutput.bWork;


_i:=E_Cylinder.UnloadFrockConveyorPush;
G_arrCylinder[_i].stInput.bHome:=GVL.I.bUnloadFrockConveyorPush_Cyl_H;
G_arrCylinder[_i].stInput.bWork:=GVL.I.bUnloadFrockConveyorPush_Cyl_W;
GVL.Q.bUnloadFrockConveyorPush_Cyl_H:=G_arrCylinder[_i].stOutput.bHome;
GVL.Q.bUnloadFrockConveyorPush_Cyl_W:=G_arrCylinder[_i].stOutput.bWork;

_i:=E_Cylinder.OpenLockElevator;
G_arrCylinder[_i].stInput.bHome:=GVL.I.bOpenLockElevator_Cyl_H;
G_arrCylinder[_i].stInput.bWork:=GVL.I.bOpenLockElevator_Cyl_W;
GVL.Q.bOpenLockElevator_Cyl_H:=G_arrCylinder[_i].stOutput.bHome;
GVL.Q.bOpenLockElevator_Cyl_W:=G_arrCylinder[_i].stOutput.bWork;

_i:=E_Cylinder.OpenLockPin;
G_arrCylinder[_i].stInput.bHome:=NOT GVL.I.bOpenLockPin_Cyl_W;
G_arrCylinder[_i].stInput.bWork:=GVL.I.bOpenLockPin_Cyl_W;
GVL.Q.bOpenLockPin_Cyl_H:=G_arrCylinder[_i].stOutput.bHome;
GVL.Q.bOpenLockPin_Cyl_W:=G_arrCylinder[_i].stOutput.bWork;

_i:=E_Cylinder.TakeUcElevator;
G_arrCylinder[_i].stInput.bHome:=GVL.I.bTakeUcElevator_Cyl_H;
G_arrCylinder[_i].stInput.bWork:=GVL.I.bTakeUcElevator_Cyl_W;
GVL.Q.bTakeUcElevator_Cyl_H:=G_arrCylinder[_i].stOutput.bHome;
GVL.Q.bTakeUcElevator_Cyl_W:=G_arrCylinder[_i].stOutput.bWork;

_i:=E_Cylinder.TakeUcPush1;
G_arrCylinder[_i].stInput.bHome:=GVL.I.bTakeUcPush1_Cyl_H;
G_arrCylinder[_i].stInput.bWork:=GVL.I.bTakeUcPush1_Cyl_W;
GVL.Q.bTakeUcPush1_Cyl_H:=G_arrCylinder[_i].stOutput.bHome;
GVL.Q.bTakeUcPush1_Cyl_W:=G_arrCylinder[_i].stOutput.bWork;

_i:=E_Cylinder.UnloadUcBeltTipper;
G_arrCylinder[_i].stInput.bHome:=GVL.I.bUnloadUcBeltTipper_Cyl_H;
G_arrCylinder[_i].stInput.bWork:=GVL.I.bUnloadUcBeltTipper_Cyl_W;
GVL.Q.bUnloadUcBeltTipper_Cyl_H:=G_arrCylinder[_i].stOutput.bHome;
GVL.Q.bUnloadUcBeltTipper_Cyl_W:=G_arrCylinder[_i].stOutput.bWork;

_i:=E_Cylinder.UnloadUcBeltLift;
G_arrCylinder[_i].stInput.bHome:=GVL.I.bUnloadUcBeltLift_Cyl_H;
G_arrCylinder[_i].stInput.bWork:=GVL.I.bUnloadUcBeltLift_Cyl_W;
GVL.Q.bUnloadUcBeltLift_Cyl_H:=G_arrCylinder[_i].stOutput.bHome;
GVL.Q.bUnloadUcBeltLift_Cyl_W:=G_arrCylinder[_i].stOutput.bWork;

_i:=E_Cylinder.OpenLockTranslation;
G_arrCylinder[_i].stInput.bHome:=GVL.I.bOpenLockTranslation_Cyl_H;
G_arrCylinder[_i].stInput.bWork:=GVL.I.bOpenLockTranslation_Cyl_W;
GVL.Q.bOpenLockTranslation_Cyl_H:=G_arrCylinder[_i].stOutput.bHome;
GVL.Q.bOpenLockTranslation_Cyl_W:=G_arrCylinder[_i].stOutput.bWork;

_i:=E_Cylinder.TakeUcFrockClamp;
G_arrCylinder[_i].stInput.bHome:=G_arrCylinder[_i].stOutput.bHome;
G_arrCylinder[_i].stInput.bWork:=G_arrCylinder[_i].stOutput.bWork;
GVL.Q.bTakeUcFrockClamp_Cyl_H:=G_arrCylinder[_i].stOutput.bHome;
GVL.Q.bTakeUcFrockClamp_Cyl_W:=G_arrCylinder[_i].stOutput.bWork;

_i:=E_Cylinder.OpenLockPressPush;
G_arrCylinder[_i].stInput.bHome:=GVL.I.bOpenLockPressPush_Cyl_H;
G_arrCylinder[_i].stInput.bWork:=GVL.I.bOpenLockPressPush_Cyl_W;
GVL.Q.bOpenLockPressPush_Cyl_H:=G_arrCylinder[_i].stOutput.bHome;
GVL.Q.bOpenLockPressPush_Cyl_W:=G_arrCylinder[_i].stOutput.bWork;

_i:=E_Cylinder.OpenLockPressRotate;
G_arrCylinder[_i].stInput.bHome:=GVL.I.bOpenLockPressRotate_Cyl_H;
G_arrCylinder[_i].stInput.bWork:=GVL.I.bOpenLockPressRotate_Cyl_W;
GVL.Q.bOpenLockPressRotate_Cyl_H:=G_arrCylinder[_i].stOutput.bHome;
GVL.Q.bOpenLockPressRotate_Cyl_W:=G_arrCylinder[_i].stOutput.bWork;

_i:=E_Cylinder.AcquirePrevent2;
G_arrCylinder[_i].stInput.bHome:=GVL.I.bAcquirePrevent2_Cyl_H;
G_arrCylinder[_i].stInput.bWork:=GVL.I.bAcquirePrevent2_Cyl_W;
GVL.Q.bAcquirePrevent2_Cyl_H:=G_arrCylinder[_i].stOutput.bHome;
GVL.Q.bAcquirePrevent2_Cyl_W:=G_arrCylinder[_i].stOutput.bWork;

_i:=E_Cylinder.Line0PushElevator;
G_arrCylinder[_i].stInput.bHome:=GVL.I.bLine0PushElevator_Cyl_H;
G_arrCylinder[_i].stInput.bWork:=GVL.I.bLine0PushElevator_Cyl_W;
GVL.Q.bLine0PushElevator_Cyl_H:=G_arrCylinder[_i].stOutput.bHome;
GVL.Q.bLine0PushElevator_Cyl_W:=G_arrCylinder[_i].stOutput.bWork;
END_ACTION

ACTION A_CylinderTest:
FOR _i:=0 TO 50 BY 1 DO
	G_arrCylinder[_i].ID:=TO_BYTE(_i+50);
	_arrCylTon_H[_i](IN:=G_arrCylinder[_i].stOutput.bHome , PT:=T#2S , Q=> , ET=> );
	_arrCylTon_W[_i](IN:=G_arrCylinder[_i].stOutput.bWork , PT:=T#2S , Q=> , ET=> );
	G_arrCylinder[_i].stInput.bHome:=_arrCylTon_H[_i].Q;
	G_arrCylinder[_i].stInput.bWork:=_arrCylTon_W[_i].Q;
END_FOR

_i:=E_Cylinder.Line0Part;
GVL.Q.bLine0Part_Cyl_H:=G_arrCylinder[_i].stOutput.bHome;
GVL.Q.bLine0Part_Cyl_W:=G_arrCylinder[_i].stOutput.bWork;

_i:=E_Cylinder.Line0Prevent;
GVL.Q.bLine0Prevent_Cyl_H:=G_arrCylinder[_i].stOutput.bHome;
GVL.Q.bLine0Prevent_Cyl_W:=G_arrCylinder[_i].stOutput.bWork;

_i:=E_Cylinder.Line0Push;
GVL.Q.bLine0Push_Cyl_H:=G_arrCylinder[_i].stOutput.bHome;
GVL.Q.bLine0Push_Cyl_W:=G_arrCylinder[_i].stOutput.bWork;

_i:=E_Cylinder.AcquirePrevent0;
GVL.Q.bAcquirePrevent0_Cyl_H:=G_arrCylinder[_i].stOutput.bHome;
GVL.Q.bAcquirePrevent0_Cyl_W:=G_arrCylinder[_i].stOutput.bWork;

_i:=E_Cylinder.AcquirePrevent1;
GVL.Q.bAcquirePrevent1_Cyl_H:=G_arrCylinder[_i].stOutput.bHome;
GVL.Q.bAcquirePrevent1_Cyl_W:=G_arrCylinder[_i].stOutput.bWork;

_i:=E_Cylinder.AcquireLift;
GVL.Q.bAcquireLift_Cyl_H:=G_arrCylinder[_i].stOutput.bHome;
GVL.Q.bAcquireLift_Cyl_W:=G_arrCylinder[_i].stOutput.bWork;

_i:=E_Cylinder.AcquirePush;
GVL.Q.bAcquirePush_Cyl_H:=G_arrCylinder[_i].stOutput.bHome;
GVL.Q.bAcquirePush_Cyl_W:=G_arrCylinder[_i].stOutput.bWork;

_i:=E_Cylinder.AcquireElevator;
GVL.Q.bAcquireElevator_Cyl_H:=G_arrCylinder[_i].stOutput.bHome;
GVL.Q.bAcquireElevator_Cyl_W:=G_arrCylinder[_i].stOutput.bWork;

_i:=E_Cylinder.SteeringLift;
GVL.Q.bSteeringLift_Cyl_H:=G_arrCylinder[_i].stOutput.bHome;
GVL.Q.bSteeringLift_Cyl_W:=G_arrCylinder[_i].stOutput.bWork;

_i:=E_Cylinder.SteeringAcquireElevator;
GVL.Q.bSteeringAcquireElevator_Cyl_H:=G_arrCylinder[_i].stOutput.bHome;
GVL.Q.bSteeringAcquireElevator_Cyl_W:=G_arrCylinder[_i].stOutput.bWork;

_i:=E_Cylinder.SteeringRotate;
GVL.Q.bSteeringRotate_Cyl_H:=G_arrCylinder[_i].stOutput.bHome;
GVL.Q.bSteeringRotate_Cyl_W:=G_arrCylinder[_i].stOutput.bWork;

_i:=E_Cylinder.SteeringAcquireLimit;
GVL.Q.bSteeringAcquireLimit_Cyl_H:=G_arrCylinder[_i].stOutput.bHome;
GVL.Q.bSteeringAcquireLimit_Cyl_W:=G_arrCylinder[_i].stOutput.bWork;

_i:=E_Cylinder.OpenLockPrevent;
GVL.Q.bOpenLockPrevent_Cyl_H:=G_arrCylinder[_i].stOutput.bHome;
GVL.Q.bOpenLockPrevent_Cyl_W:=G_arrCylinder[_i].stOutput.bWork;

_i:=E_Cylinder.OpenLockLift;
GVL.Q.bOpenLockLift_Cyl_H:=G_arrCylinder[_i].stOutput.bHome;
GVL.Q.bOpenLockLift_Cyl_W:=G_arrCylinder[_i].stOutput.bWork;

_i:=E_Cylinder.OpenLockPush;
GVL.Q.bOpenLockPush_Cyl_H:=G_arrCylinder[_i].stOutput.bHome;
GVL.Q.bOpenLockPush_Cyl_W:=G_arrCylinder[_i].stOutput.bWork;

_i:=E_Cylinder.OpenLockRotate;
GVL.Q.bOpenLockRotate_Cyl_H:=G_arrCylinder[_i].stOutput.bHome;
GVL.Q.bOpenLockRotate_Cyl_W:=G_arrCylinder[_i].stOutput.bWork;

_i:=E_Cylinder.OpenLockPush2;
GVL.Q.bOpenLockPush2_Cyl_H:=G_arrCylinder[_i].stOutput.bHome;
GVL.Q.bOpenLockPush2_Cyl_W:=G_arrCylinder[_i].stOutput.bWork;

_i:=E_Cylinder.TakeUcPrevent;
GVL.Q.bTakeUcPrevent_Cyl_H:=G_arrCylinder[_i].stOutput.bHome;
GVL.Q.bTakeUcPrevent_Cyl_W:=G_arrCylinder[_i].stOutput.bWork;

_i:=E_Cylinder.TakeUcLift;
GVL.Q.bTakeUcLift_Cyl_H:=G_arrCylinder[_i].stOutput.bHome;
GVL.Q.bTakeUcLift_Cyl_W:=G_arrCylinder[_i].stOutput.bWork;

_i:=E_Cylinder.TakeUcPush;
GVL.Q.bTakeUcPush_Cyl_H:=G_arrCylinder[_i].stOutput.bHome;
GVL.Q.bTakeUcPush_Cyl_W:=G_arrCylinder[_i].stOutput.bWork;

_i:=E_Cylinder.TakeUcRotate;
GVL.Q.bTakeUcRotate_Cyl_H:=G_arrCylinder[_i].stOutput.bHome;
GVL.Q.bTakeUcRotate_Cyl_W:=G_arrCylinder[_i].stOutput.bWork;

_i:=E_Cylinder.TakeUcStandard;
GVL.Q.bTakeUcStandard_Cyl_H:=G_arrCylinder[_i].stOutput.bHome;
GVL.Q.bTakeUcStandard_Cyl_W:=G_arrCylinder[_i].stOutput.bWork;

_i:=E_Cylinder.UnloadFrockPrevent;
GVL.Q.bUnloadFrockPrevent_Cyl_H:=G_arrCylinder[_i].stOutput.bHome;
GVL.Q.bUnloadFrockPrevent_Cyl_W:=G_arrCylinder[_i].stOutput.bWork;

_i:=E_Cylinder.UnloadFrockLift;
GVL.Q.bUnloadFrockLift_Cyl_H:=G_arrCylinder[_i].stOutput.bHome;
GVL.Q.bUnloadFrockLift_Cyl_W:=G_arrCylinder[_i].stOutput.bWork;

_i:=E_Cylinder.UnloadFrockPush;
GVL.Q.bUnloadFrockPush_Cyl_H:=G_arrCylinder[_i].stOutput.bHome;
GVL.Q.bUnloadFrockPush_Cyl_W:=G_arrCylinder[_i].stOutput.bWork;

_i:=E_Cylinder.TakeUc1Y;
GVL.Q.bTakeUc1Y_Cyl_H:=G_arrCylinder[_i].stOutput.bHome;
GVL.Q.bTakeUc1Y_Cyl_W:=G_arrCylinder[_i].stOutput.bWork;

_i:=E_Cylinder.TakeUc1Z1;
GVL.Q.bTakeUc1Z1_Cyl_H:=G_arrCylinder[_i].stOutput.bHome;
GVL.Q.bTakeUc1Z1_Cyl_W:=G_arrCylinder[_i].stOutput.bWork;

_i:=E_Cylinder.TakeUc1Z2;
GVL.Q.bTakeUc1Z2_Cyl_H:=G_arrCylinder[_i].stOutput.bHome;
GVL.Q.bTakeUc1Z2_Cyl_W:=G_arrCylinder[_i].stOutput.bWork;

_i:=E_Cylinder.TakeUc1Rotate;
GVL.Q.bTakeUc1Rotate_Cyl_H:=G_arrCylinder[_i].stOutput.bHome;
GVL.Q.bTakeUc1Rotate_Cyl_W:=G_arrCylinder[_i].stOutput.bWork;

_i:=E_Cylinder.TakeUc1Clamp;
GVL.Q.bTakeUc1Clamp_Cyl_H:=G_arrCylinder[_i].stOutput.bHome;
GVL.Q.bTakeUc1Clamp_Cyl_W:=G_arrCylinder[_i].stOutput.bWork;

_i:=E_Cylinder.UnloadUcElevator;
GVL.Q.bUnloadUcElevator_Cyl_H:=G_arrCylinder[_i].stOutput.bHome;
GVL.Q.bUnloadUcElevator_Cyl_W:=G_arrCylinder[_i].stOutput.bWork;

_i:=E_Cylinder.UnloadUcConveyorPush;
GVL.Q.bUnloadUcConveyorPush_Cyl_H:=G_arrCylinder[_i].stOutput.bHome;
GVL.Q.bUnloadUcConveyorPush_Cyl_W:=G_arrCylinder[_i].stOutput.bWork;

_i:=E_Cylinder.UnloadFrockConveyorPrevent;
GVL.Q.bUnloadFrockConveyorPrevent_Cyl_H:=G_arrCylinder[_i].stOutput.bHome;
GVL.Q.bUnloadFrockConveyorPrevent_Cyl_W:=G_arrCylinder[_i].stOutput.bWork;

_i:=E_Cylinder.UnloadFrockConveyorPush;
GVL.Q.bUnloadFrockConveyorPush_Cyl_H:=G_arrCylinder[_i].stOutput.bHome;
GVL.Q.bUnloadFrockConveyorPush_Cyl_W:=G_arrCylinder[_i].stOutput.bWork;

_i:=E_Cylinder.OpenLockElevator;
GVL.Q.bOpenLockElevator_Cyl_H:=G_arrCylinder[_i].stOutput.bHome;
GVL.Q.bOpenLockElevator_Cyl_W:=G_arrCylinder[_i].stOutput.bWork;

_i:=E_Cylinder.OpenLockPin;
GVL.Q.bOpenLockPin_Cyl_H:=G_arrCylinder[_i].stOutput.bHome;
GVL.Q.bOpenLockPin_Cyl_W:=G_arrCylinder[_i].stOutput.bWork;

_i:=E_Cylinder.TakeUcElevator;
GVL.Q.bTakeUcElevator_Cyl_H:=G_arrCylinder[_i].stOutput.bHome;
GVL.Q.bTakeUcElevator_Cyl_W:=G_arrCylinder[_i].stOutput.bWork;

_i:=E_Cylinder.TakeUcPush1;
GVL.Q.bTakeUcPush1_Cyl_H:=G_arrCylinder[_i].stOutput.bHome;
GVL.Q.bTakeUcPush1_Cyl_W:=G_arrCylinder[_i].stOutput.bWork;


_i:=E_Cylinder.UnloadUcBeltTipper;
GVL.Q.bUnloadUcBeltTipper_Cyl_H:=G_arrCylinder[_i].stOutput.bHome;
GVL.Q.bUnloadUcBeltTipper_Cyl_W:=G_arrCylinder[_i].stOutput.bWork;

_i:=E_Cylinder.UnloadUcBeltLift;
GVL.Q.bUnloadUcBeltLift_Cyl_H:=G_arrCylinder[_i].stOutput.bHome;
GVL.Q.bUnloadUcBeltLift_Cyl_W:=G_arrCylinder[_i].stOutput.bWork;

_i:=E_Cylinder.OpenLockTranslation;
GVL.Q.bOpenLockTranslation_Cyl_H:=G_arrCylinder[_i].stOutput.bHome;
GVL.Q.bOpenLockTranslation_Cyl_W:=G_arrCylinder[_i].stOutput.bWork;

_i:=E_Cylinder.TakeUcFrockClamp;
GVL.Q.bTakeUcFrockClamp_Cyl_H:=G_arrCylinder[_i].stOutput.bHome;
GVL.Q.bTakeUcFrockClamp_Cyl_W:=G_arrCylinder[_i].stOutput.bWork;

_i:=E_Cylinder.OpenLockPressPush;
GVL.Q.bOpenLockPressPush_Cyl_H:=G_arrCylinder[_i].stOutput.bHome;
GVL.Q.bOpenLockPressPush_Cyl_W:=G_arrCylinder[_i].stOutput.bWork;

_i:=E_Cylinder.OpenLockPressRotate;
GVL.Q.bOpenLockPressRotate_Cyl_H:=G_arrCylinder[_i].stOutput.bHome;
GVL.Q.bOpenLockPressRotate_Cyl_W:=G_arrCylinder[_i].stOutput.bWork;

_i:=E_Cylinder.AcquirePrevent2;
GVL.Q.bAcquirePrevent2_Cyl_H:=G_arrCylinder[_i].stOutput.bHome;
GVL.Q.bAcquirePrevent2_Cyl_W:=G_arrCylinder[_i].stOutput.bWork;

_i:=E_Cylinder.Line0PushElevator;
GVL.Q.bLine0PushElevator_Cyl_H:=G_arrCylinder[_i].stOutput.bHome;
GVL.Q.bLine0PushElevator_Cyl_W:=G_arrCylinder[_i].stOutput.bWork;
END_ACTION

ACTION A_CylinderTest069:
FOR _i:=0 TO 50 BY 1 DO
	G_arrCylinder[_i].ID:=TO_BYTE(_i+50);
	_arrCylTon_H[_i](IN:=G_arrCylinder[_i].stOutput.bHome , PT:=T#2S , Q=> , ET=> );
	_arrCylTon_W[_i](IN:=G_arrCylinder[_i].stOutput.bWork , PT:=T#2S , Q=> , ET=> );
	G_arrCylinder[_i].stInput.bHome:=_arrCylTon_H[_i].Q;
	G_arrCylinder[_i].stInput.bWork:=_arrCylTon_W[_i].Q;
END_FOR

_i:=E_Cylinder.Line0Part;
GVL.Q.bLine0Part_Cyl_H:=G_arrCylinder[_i].stOutput.bHome;
GVL.Q.bLine0Part_Cyl_W:=G_arrCylinder[_i].stOutput.bWork;

_i:=E_Cylinder.Line0Prevent;
GVL.Q.bLine0Prevent_Cyl_H:=G_arrCylinder[_i].stOutput.bHome;
GVL.Q.bLine0Prevent_Cyl_W:=G_arrCylinder[_i].stOutput.bWork;

_i:=E_Cylinder.Line0Push;
GVL.Q.bLine0Push_Cyl_H:=G_arrCylinder[_i].stOutput.bHome;
GVL.Q.bLine0Push_Cyl_W:=G_arrCylinder[_i].stOutput.bWork;

_i:=E_Cylinder.AcquirePrevent0;
G_arrCylinder[_i].stInput.bWork:=GVL.I.bAcquirePrevent0_Cyl_W;
GVL.Q.bAcquirePrevent0_Cyl_H:=G_arrCylinder[_i].stOutput.bHome;
GVL.Q.bAcquirePrevent0_Cyl_W:=G_arrCylinder[_i].stOutput.bWork;

_i:=E_Cylinder.AcquirePrevent1;
G_arrCylinder[_i].stInput.bWork:=GVL.I.bAcquirePrevent1_Cyl_W;
GVL.Q.bAcquirePrevent1_Cyl_H:=G_arrCylinder[_i].stOutput.bHome;
GVL.Q.bAcquirePrevent1_Cyl_W:=G_arrCylinder[_i].stOutput.bWork;

_i:=E_Cylinder.AcquireLift;
G_arrCylinder[_i].stInput.bHome:=GVL.I.bAcquireLift_Cyl_H;
G_arrCylinder[_i].stInput.bWork:=GVL.I.bAcquireLift_Cyl_W;
GVL.Q.bAcquireLift_Cyl_H:=G_arrCylinder[_i].stOutput.bHome;
GVL.Q.bAcquireLift_Cyl_W:=G_arrCylinder[_i].stOutput.bWork;

_i:=E_Cylinder.AcquirePush;
G_arrCylinder[_i].stInput.bHome:=GVL.I.bAcquirePush_Cyl_H;
G_arrCylinder[_i].stInput.bWork:=GVL.I.bAcquirePush_Cyl_W;
GVL.Q.bAcquirePush_Cyl_H:=G_arrCylinder[_i].stOutput.bHome;
GVL.Q.bAcquirePush_Cyl_W:=G_arrCylinder[_i].stOutput.bWork;

_i:=E_Cylinder.AcquireElevator;
G_arrCylinder[_i].stInput.bHome:=GVL.I.bAcquireElevator_Cyl_H;
G_arrCylinder[_i].stInput.bWork:=GVL.I.bAcquireElevator_Cyl_W;
GVL.Q.bAcquireElevator_Cyl_H:=G_arrCylinder[_i].stOutput.bHome;
GVL.Q.bAcquireElevator_Cyl_W:=G_arrCylinder[_i].stOutput.bWork;

_i:=E_Cylinder.SteeringLift;
G_arrCylinder[_i].stInput.bHome:=GVL.I.bSteeringLift_Cyl_H;
G_arrCylinder[_i].stInput.bWork:=GVL.I.bSteeringLift_Cyl_W;
GVL.Q.bSteeringLift_Cyl_H:=G_arrCylinder[_i].stOutput.bHome;
GVL.Q.bSteeringLift_Cyl_W:=G_arrCylinder[_i].stOutput.bWork;

_i:=E_Cylinder.SteeringAcquireElevator;
G_arrCylinder[_i].stInput.bHome:=GVL.I.bSteeringAcquireElevator_Cyl_H;
G_arrCylinder[_i].stInput.bWork:=GVL.I.bSteeringAcquireElevator_Cyl_W;
GVL.Q.bSteeringAcquireElevator_Cyl_H:=G_arrCylinder[_i].stOutput.bHome;
GVL.Q.bSteeringAcquireElevator_Cyl_W:=G_arrCylinder[_i].stOutput.bWork;

_i:=E_Cylinder.SteeringRotate;
G_arrCylinder[_i].stInput.bHome:=GVL.I.bSteeringRotate_Cyl_H;
G_arrCylinder[_i].stInput.bWork:=GVL.I.bSteeringRotate_Cyl_W;
GVL.Q.bSteeringRotate_Cyl_H:=G_arrCylinder[_i].stOutput.bHome;
GVL.Q.bSteeringRotate_Cyl_W:=G_arrCylinder[_i].stOutput.bWork;

_i:=E_Cylinder.SteeringAcquireLimit;
G_arrCylinder[_i].stInput.bHome:=GVL.I.bSteeringAcquireLimit_Cyl_H;
G_arrCylinder[_i].stInput.bWork:=GVL.I.bSteeringAcquireLimit_Cyl_W;
GVL.Q.bSteeringAcquireLimit_Cyl_H:=G_arrCylinder[_i].stOutput.bHome;
GVL.Q.bSteeringAcquireLimit_Cyl_W:=G_arrCylinder[_i].stOutput.bWork;

_i:=E_Cylinder.OpenLockPrevent;
G_arrCylinder[_i].stInput.bWork:=GVL.I.bOpenLockPrevent_Cyl_W;
GVL.Q.bOpenLockPrevent_Cyl_H:=G_arrCylinder[_i].stOutput.bHome;
GVL.Q.bOpenLockPrevent_Cyl_W:=G_arrCylinder[_i].stOutput.bWork;

_i:=E_Cylinder.OpenLockLift;
G_arrCylinder[_i].stInput.bHome:=GVL.I.bOpenLockLift_Cyl_H;
G_arrCylinder[_i].stInput.bWork:=GVL.I.bOpenLockLift_Cyl_W;
GVL.Q.bOpenLockLift_Cyl_H:=G_arrCylinder[_i].stOutput.bHome;
GVL.Q.bOpenLockLift_Cyl_W:=G_arrCylinder[_i].stOutput.bWork;

_i:=E_Cylinder.OpenLockPush;
G_arrCylinder[_i].stInput.bHome:=GVL.I.bOpenLockPush_Cyl_H;
G_arrCylinder[_i].stInput.bWork:=GVL.I.bOpenLockPush_Cyl_W;
GVL.Q.bOpenLockPush_Cyl_H:=G_arrCylinder[_i].stOutput.bHome;
GVL.Q.bOpenLockPush_Cyl_W:=G_arrCylinder[_i].stOutput.bWork;

_i:=E_Cylinder.OpenLockRotate;
G_arrCylinder[_i].stInput.bHome:=GVL.I.bOpenLockRotate_Cyl_H;
G_arrCylinder[_i].stInput.bWork:=GVL.I.bOpenLockRotate_Cyl_W;
GVL.Q.bOpenLockRotate_Cyl_H:=G_arrCylinder[_i].stOutput.bHome;
GVL.Q.bOpenLockRotate_Cyl_W:=G_arrCylinder[_i].stOutput.bWork;

_i:=E_Cylinder.OpenLockPush2;
//G_arrCylinder[_i].stInput.bHome:=GVL.I.bOpenLockPush2_Cyl_H;
G_arrCylinder[_i].stInput.bHome:=NOT GVL.I.bOpenLockPush2_Cyl_W;
G_arrCylinder[_i].stInput.bWork:=GVL.I.bOpenLockPush2_Cyl_W;
GVL.Q.bOpenLockPush2_Cyl_H:=G_arrCylinder[_i].stOutput.bHome;
GVL.Q.bOpenLockPush2_Cyl_W:=G_arrCylinder[_i].stOutput.bWork;

_i:=E_Cylinder.TakeUcPrevent;
G_arrCylinder[_i].stInput.bWork:=GVL.I.bTakeUcPrevent_Cyl_W;
GVL.Q.bTakeUcPrevent_Cyl_H:=G_arrCylinder[_i].stOutput.bHome;
GVL.Q.bTakeUcPrevent_Cyl_W:=G_arrCylinder[_i].stOutput.bWork;

_i:=E_Cylinder.TakeUcLift;
G_arrCylinder[_i].stInput.bHome:=GVL.I.bTakeUcLift_Cyl_H;
G_arrCylinder[_i].stInput.bWork:=GVL.I.bTakeUcLift_Cyl_W;
GVL.Q.bTakeUcLift_Cyl_H:=G_arrCylinder[_i].stOutput.bHome;
GVL.Q.bTakeUcLift_Cyl_W:=G_arrCylinder[_i].stOutput.bWork;

_i:=E_Cylinder.TakeUcPush;
G_arrCylinder[_i].stInput.bHome:=GVL.I.bTakeUcPush_Cyl_H;
G_arrCylinder[_i].stInput.bWork:=GVL.I.bTakeUcPush_Cyl_W;
GVL.Q.bTakeUcPush_Cyl_H:=G_arrCylinder[_i].stOutput.bHome;
GVL.Q.bTakeUcPush_Cyl_W:=G_arrCylinder[_i].stOutput.bWork;

_i:=E_Cylinder.TakeUcRotate;
G_arrCylinder[_i].stInput.bHome:=GVL.I.bTakeUcRotate_Cyl_H;
G_arrCylinder[_i].stInput.bWork:=GVL.I.bTakeUcRotate_Cyl_W;
GVL.Q.bTakeUcRotate_Cyl_H:=G_arrCylinder[_i].stOutput.bHome;
GVL.Q.bTakeUcRotate_Cyl_W:=G_arrCylinder[_i].stOutput.bWork;

_i:=E_Cylinder.TakeUcStandard;
G_arrCylinder[_i].stInput.bHome:=GVL.I.bTakeUcStandard_Cyl_H;
G_arrCylinder[_i].stInput.bWork:=GVL.I.bTakeUcStandard_Cyl_W;
GVL.Q.bTakeUcStandard_Cyl_H:=G_arrCylinder[_i].stOutput.bHome;
GVL.Q.bTakeUcStandard_Cyl_W:=G_arrCylinder[_i].stOutput.bWork;

_i:=E_Cylinder.UnloadFrockPrevent;
G_arrCylinder[_i].stInput.bHome:=GVL.I.bUnloadFrockPrevent_Cyl_H;
G_arrCylinder[_i].stInput.bWork:=GVL.I.bUnloadFrockPrevent_Cyl_W;
GVL.Q.bUnloadFrockPrevent_Cyl_H:=G_arrCylinder[_i].stOutput.bHome;
GVL.Q.bUnloadFrockPrevent_Cyl_W:=G_arrCylinder[_i].stOutput.bWork;

_i:=E_Cylinder.UnloadFrockLift;
G_arrCylinder[_i].stInput.bHome:=GVL.I.bUnloadFrockLift_Cyl_H;
G_arrCylinder[_i].stInput.bWork:=GVL.I.bUnloadFrockLift_Cyl_W;
GVL.Q.bUnloadFrockLift_Cyl_H:=G_arrCylinder[_i].stOutput.bHome;
GVL.Q.bUnloadFrockLift_Cyl_W:=G_arrCylinder[_i].stOutput.bWork;

_i:=E_Cylinder.UnloadFrockPush;
G_arrCylinder[_i].stInput.bHome:=GVL.I.bUnloadFrockPush_Cyl_H;
G_arrCylinder[_i].stInput.bWork:=GVL.I.bUnloadFrockPush_Cyl_W;
GVL.Q.bUnloadFrockPush_Cyl_H:=G_arrCylinder[_i].stOutput.bHome;
GVL.Q.bUnloadFrockPush_Cyl_W:=G_arrCylinder[_i].stOutput.bWork;

_i:=E_Cylinder.TakeUc1Y;
G_arrCylinder[_i].stInput.bHome:=GVL.I.bTakeUc1Y_Cyl_H;
G_arrCylinder[_i].stInput.bWork:=GVL.I.bTakeUc1Y_Cyl_W;
GVL.Q.bTakeUc1Y_Cyl_H:=G_arrCylinder[_i].stOutput.bHome;
GVL.Q.bTakeUc1Y_Cyl_W:=G_arrCylinder[_i].stOutput.bWork;

_i:=E_Cylinder.TakeUc1Z1;
G_arrCylinder[_i].stInput.bHome:=GVL.I.bTakeUc1Z1_Cyl_H;
G_arrCylinder[_i].stInput.bWork:=GVL.I.bTakeUc1Z1_Cyl_W;
GVL.Q.bTakeUc1Z1_Cyl_H:=G_arrCylinder[_i].stOutput.bHome;
GVL.Q.bTakeUc1Z1_Cyl_W:=G_arrCylinder[_i].stOutput.bWork;

_i:=E_Cylinder.TakeUc1Z2;
G_arrCylinder[_i].stInput.bHome:=GVL.I.bTakeUc1Z2_Cyl_H;
G_arrCylinder[_i].stInput.bWork:=GVL.I.bTakeUc1Z2_Cyl_W;
GVL.Q.bTakeUc1Z2_Cyl_H:=G_arrCylinder[_i].stOutput.bHome;
GVL.Q.bTakeUc1Z2_Cyl_W:=G_arrCylinder[_i].stOutput.bWork;

_i:=E_Cylinder.TakeUc1Rotate;
G_arrCylinder[_i].stInput.bHome:=GVL.I.bTakeUc1Rotate_Cyl_H;
G_arrCylinder[_i].stInput.bWork:=GVL.I.bTakeUc1Rotate_Cyl_W;
GVL.Q.bTakeUc1Rotate_Cyl_H:=G_arrCylinder[_i].stOutput.bHome;
GVL.Q.bTakeUc1Rotate_Cyl_W:=G_arrCylinder[_i].stOutput.bWork;

_i:=E_Cylinder.TakeUc1Clamp;
G_arrCylinder[_i].stInput.bHome:=GVL.I.bTakeUc1Clamp_Cyl_H;
//G_arrCylinder[_i].stInput.bWork:=GVL.I.bTakeUc1Clamp_Cyl_W;
GVL.Q.bTakeUc1Clamp_Cyl_H:=G_arrCylinder[_i].stOutput.bHome;
GVL.Q.bTakeUc1Clamp_Cyl_W:=G_arrCylinder[_i].stOutput.bWork;

_i:=E_Cylinder.UnloadUcElevator;
//G_arrCylinder[_i].stInput.bHome:=GVL.I.bUnloadUcElevator_Cyl_H;
//G_arrCylinder[_i].stInput.bWork:=GVL.I.bUnloadUcElevator_Cyl_W;
GVL.Q.bUnloadUcElevator_Cyl_H:=G_arrCylinder[_i].stOutput.bHome;
GVL.Q.bUnloadUcElevator_Cyl_W:=G_arrCylinder[_i].stOutput.bWork;

_i:=E_Cylinder.UnloadUcConveyorPush;
//G_arrCylinder[_i].stInput.bHome:=GVL.I.bUnloadUcConveyorPush_Cyl_H;
//G_arrCylinder[_i].stInput.bWork:=GVL.I.bUnloadUcConveyorPush_Cyl_W;
GVL.Q.bUnloadUcConveyorPush_Cyl_H:=G_arrCylinder[_i].stOutput.bHome;
GVL.Q.bUnloadUcConveyorPush_Cyl_W:=G_arrCylinder[_i].stOutput.bWork;

_i:=E_Cylinder.UnloadFrockConveyorPrevent;
//G_arrCylinder[_i].stInput.bHome:=GVL.I.bUnloadFrockConveyorPrevent_Cyl_H;
//G_arrCylinder[_i].stInput.bWork:=GVL.I.bUnloadFrockConveyorPrevent_Cyl_W;
GVL.Q.bUnloadFrockConveyorPrevent_Cyl_H:=G_arrCylinder[_i].stOutput.bHome;
GVL.Q.bUnloadFrockConveyorPrevent_Cyl_W:=G_arrCylinder[_i].stOutput.bWork;

_i:=E_Cylinder.UnloadFrockConveyorPush;
//G_arrCylinder[_i].stInput.bHome:=GVL.I.bUnloadFrockConveyorPush_Cyl_H;
//G_arrCylinder[_i].stInput.bWork:=GVL.I.bUnloadFrockConveyorPush_Cyl_W;
GVL.Q.bUnloadFrockConveyorPush_Cyl_H:=G_arrCylinder[_i].stOutput.bHome;
GVL.Q.bUnloadFrockConveyorPush_Cyl_W:=G_arrCylinder[_i].stOutput.bWork;

_i:=E_Cylinder.OpenLockElevator;
G_arrCylinder[_i].stInput.bHome:=GVL.I.bOpenLockElevator_Cyl_H;
G_arrCylinder[_i].stInput.bWork:=GVL.I.bOpenLockElevator_Cyl_W;
GVL.Q.bOpenLockElevator_Cyl_H:=G_arrCylinder[_i].stOutput.bHome;
GVL.Q.bOpenLockElevator_Cyl_W:=G_arrCylinder[_i].stOutput.bWork;

_i:=E_Cylinder.OpenLockPin;
G_arrCylinder[_i].stInput.bHome:=GVL.I.bOpenLockPin_Cyl_H;
G_arrCylinder[_i].stInput.bWork:=GVL.I.bOpenLockPin_Cyl_W;
GVL.Q.bOpenLockPin_Cyl_H:=G_arrCylinder[_i].stOutput.bHome;
GVL.Q.bOpenLockPin_Cyl_W:=G_arrCylinder[_i].stOutput.bWork;

_i:=E_Cylinder.TakeUcElevator;
G_arrCylinder[_i].stInput.bHome:=GVL.I.bTakeUcElevator_Cyl_H;
G_arrCylinder[_i].stInput.bWork:=GVL.I.bTakeUcElevator_Cyl_W;
GVL.Q.bTakeUcElevator_Cyl_H:=G_arrCylinder[_i].stOutput.bHome;
GVL.Q.bTakeUcElevator_Cyl_W:=G_arrCylinder[_i].stOutput.bWork;

_i:=E_Cylinder.TakeUcPush1;
G_arrCylinder[_i].stInput.bHome:=GVL.I.bTakeUcPush1_Cyl_H;
G_arrCylinder[_i].stInput.bWork:=GVL.I.bTakeUcPush1_Cyl_W;
GVL.Q.bTakeUcPush1_Cyl_H:=G_arrCylinder[_i].stOutput.bHome;
GVL.Q.bTakeUcPush1_Cyl_W:=G_arrCylinder[_i].stOutput.bWork;

_i:=E_Cylinder.UnloadUcBeltTipper;
G_arrCylinder[_i].stInput.bHome:=GVL.I.bUnloadUcBeltTipper_Cyl_H;
G_arrCylinder[_i].stInput.bWork:=GVL.I.bUnloadUcBeltTipper_Cyl_W;
GVL.Q.bUnloadUcBeltTipper_Cyl_H:=G_arrCylinder[_i].stOutput.bHome;
GVL.Q.bUnloadUcBeltTipper_Cyl_W:=G_arrCylinder[_i].stOutput.bWork;

_i:=E_Cylinder.UnloadUcBeltLift;
G_arrCylinder[_i].stInput.bHome:=GVL.I.bUnloadUcBeltLift_Cyl_H;
G_arrCylinder[_i].stInput.bWork:=GVL.I.bUnloadUcBeltLift_Cyl_W;
GVL.Q.bUnloadUcBeltLift_Cyl_H:=G_arrCylinder[_i].stOutput.bHome;
GVL.Q.bUnloadUcBeltLift_Cyl_W:=G_arrCylinder[_i].stOutput.bWork;

_i:=E_Cylinder.OpenLockTranslation;
G_arrCylinder[_i].stInput.bHome:=GVL.I.bOpenLockTranslation_Cyl_H;
G_arrCylinder[_i].stInput.bWork:=GVL.I.bOpenLockTranslation_Cyl_W;
GVL.Q.bOpenLockTranslation_Cyl_H:=G_arrCylinder[_i].stOutput.bHome;
GVL.Q.bOpenLockTranslation_Cyl_W:=G_arrCylinder[_i].stOutput.bWork;

_i:=E_Cylinder.TakeUcFrockClamp;
G_arrCylinder[_i].stInput.bHome:=GVL.I.bTakeUcFrockClamp_Cyl_H;
G_arrCylinder[_i].stInput.bWork:=GVL.I.bTakeUcFrockClamp_Cyl_W;
GVL.Q.bTakeUcFrockClamp_Cyl_H:=G_arrCylinder[_i].stOutput.bHome;
GVL.Q.bTakeUcFrockClamp_Cyl_W:=G_arrCylinder[_i].stOutput.bWork;
END_ACTION

ACTION A_CylinderTest201:
FOR _i:=0 TO 50 BY 1 DO
	G_arrCylinder[_i].ID:=TO_BYTE(_i+50);
	_arrCylTon_H[_i](IN:=G_arrCylinder[_i].stOutput.bHome , PT:=T#2S , Q=> , ET=> );
	_arrCylTon_W[_i](IN:=G_arrCylinder[_i].stOutput.bWork , PT:=T#2S , Q=> , ET=> );
	G_arrCylinder[_i].stInput.bHome:=_arrCylTon_H[_i].Q;
	G_arrCylinder[_i].stInput.bWork:=_arrCylTon_W[_i].Q;
END_FOR

_i:=E_Cylinder.Line0Part;
G_arrCylinder[_i].stInput.bHome:=GVL.I.bLine0Part_Cyl_H;
G_arrCylinder[_i].stInput.bWork:=GVL.I.bLine0Part_Cyl_W;
GVL.Q.bLine0Part_Cyl_H:=G_arrCylinder[_i].stOutput.bHome;
GVL.Q.bLine0Part_Cyl_W:=G_arrCylinder[_i].stOutput.bWork;

_i:=E_Cylinder.Line0Prevent;
G_arrCylinder[_i].stInput.bHome:=GVL.I.bLine0Prevent_Cyl_H;
G_arrCylinder[_i].stInput.bWork:=GVL.I.bLine0Prevent_Cyl_W;
GVL.Q.bLine0Prevent_Cyl_H:=G_arrCylinder[_i].stOutput.bHome;
GVL.Q.bLine0Prevent_Cyl_W:=G_arrCylinder[_i].stOutput.bWork;

_i:=E_Cylinder.Line0Push;
G_arrCylinder[_i].stInput.bHome:=GVL.I.bLine0Push_Cyl_H;
G_arrCylinder[_i].stInput.bWork:=GVL.I.bLine0Push_Cyl_W;
GVL.Q.bLine0Push_Cyl_H:=G_arrCylinder[_i].stOutput.bHome;
GVL.Q.bLine0Push_Cyl_W:=G_arrCylinder[_i].stOutput.bWork;

_i:=E_Cylinder.AcquirePrevent0;
G_arrCylinder[_i].stInput.bWork:=GVL.I.bAcquirePrevent0_Cyl_W;
GVL.Q.bAcquirePrevent0_Cyl_H:=G_arrCylinder[_i].stOutput.bHome;
GVL.Q.bAcquirePrevent0_Cyl_W:=G_arrCylinder[_i].stOutput.bWork;

_i:=E_Cylinder.AcquirePrevent1;
G_arrCylinder[_i].stInput.bWork:=GVL.I.bAcquirePrevent1_Cyl_W;
GVL.Q.bAcquirePrevent1_Cyl_H:=G_arrCylinder[_i].stOutput.bHome;
GVL.Q.bAcquirePrevent1_Cyl_W:=G_arrCylinder[_i].stOutput.bWork;

_i:=E_Cylinder.AcquireLift;
G_arrCylinder[_i].stInput.bHome:=GVL.I.bAcquireLift_Cyl_H;
G_arrCylinder[_i].stInput.bWork:=GVL.I.bAcquireLift_Cyl_W;
GVL.Q.bAcquireLift_Cyl_H:=G_arrCylinder[_i].stOutput.bHome;
GVL.Q.bAcquireLift_Cyl_W:=G_arrCylinder[_i].stOutput.bWork;

_i:=E_Cylinder.AcquirePush;
G_arrCylinder[_i].stInput.bHome:=GVL.I.bAcquirePush_Cyl_H;
G_arrCylinder[_i].stInput.bWork:=GVL.I.bAcquirePush_Cyl_W;
GVL.Q.bAcquirePush_Cyl_H:=G_arrCylinder[_i].stOutput.bHome;
GVL.Q.bAcquirePush_Cyl_W:=G_arrCylinder[_i].stOutput.bWork;

_i:=E_Cylinder.AcquireElevator;
G_arrCylinder[_i].stInput.bHome:=GVL.I.bAcquireElevator_Cyl_H;
G_arrCylinder[_i].stInput.bWork:=GVL.I.bAcquireElevator_Cyl_W;
GVL.Q.bAcquireElevator_Cyl_H:=G_arrCylinder[_i].stOutput.bHome;
GVL.Q.bAcquireElevator_Cyl_W:=G_arrCylinder[_i].stOutput.bWork;

_i:=E_Cylinder.SteeringLift;
G_arrCylinder[_i].stInput.bHome:=GVL.I.bSteeringLift_Cyl_H;
G_arrCylinder[_i].stInput.bWork:=GVL.I.bSteeringLift_Cyl_W;
GVL.Q.bSteeringLift_Cyl_H:=G_arrCylinder[_i].stOutput.bHome;
GVL.Q.bSteeringLift_Cyl_W:=G_arrCylinder[_i].stOutput.bWork;

_i:=E_Cylinder.SteeringAcquireElevator;
G_arrCylinder[_i].stInput.bHome:=GVL.I.bSteeringAcquireElevator_Cyl_H;
G_arrCylinder[_i].stInput.bWork:=GVL.I.bSteeringAcquireElevator_Cyl_W;
GVL.Q.bSteeringAcquireElevator_Cyl_H:=G_arrCylinder[_i].stOutput.bHome;
GVL.Q.bSteeringAcquireElevator_Cyl_W:=G_arrCylinder[_i].stOutput.bWork;

_i:=E_Cylinder.SteeringRotate;
G_arrCylinder[_i].stInput.bHome:=GVL.I.bSteeringRotate_Cyl_H;
G_arrCylinder[_i].stInput.bWork:=GVL.I.bSteeringRotate_Cyl_W;
GVL.Q.bSteeringRotate_Cyl_H:=G_arrCylinder[_i].stOutput.bHome;
GVL.Q.bSteeringRotate_Cyl_W:=G_arrCylinder[_i].stOutput.bWork;

_i:=E_Cylinder.SteeringAcquireLimit;
G_arrCylinder[_i].stInput.bHome:=GVL.I.bSteeringAcquireLimit_Cyl_H;
G_arrCylinder[_i].stInput.bWork:=GVL.I.bSteeringAcquireLimit_Cyl_W;
GVL.Q.bSteeringAcquireLimit_Cyl_H:=G_arrCylinder[_i].stOutput.bHome;
GVL.Q.bSteeringAcquireLimit_Cyl_W:=G_arrCylinder[_i].stOutput.bWork;

_i:=E_Cylinder.OpenLockPrevent;
G_arrCylinder[_i].stInput.bWork:=GVL.I.bOpenLockPrevent_Cyl_W;
GVL.Q.bOpenLockPrevent_Cyl_H:=G_arrCylinder[_i].stOutput.bHome;
GVL.Q.bOpenLockPrevent_Cyl_W:=G_arrCylinder[_i].stOutput.bWork;

_i:=E_Cylinder.OpenLockLift;
G_arrCylinder[_i].stInput.bHome:=GVL.I.bOpenLockLift_Cyl_H;
G_arrCylinder[_i].stInput.bWork:=GVL.I.bOpenLockLift_Cyl_W;
GVL.Q.bOpenLockLift_Cyl_H:=G_arrCylinder[_i].stOutput.bHome;
GVL.Q.bOpenLockLift_Cyl_W:=G_arrCylinder[_i].stOutput.bWork;

_i:=E_Cylinder.OpenLockPush;
G_arrCylinder[_i].stInput.bHome:=GVL.I.bOpenLockPush_Cyl_H;
G_arrCylinder[_i].stInput.bWork:=GVL.I.bOpenLockPush_Cyl_W;
GVL.Q.bOpenLockPush_Cyl_H:=G_arrCylinder[_i].stOutput.bHome;
GVL.Q.bOpenLockPush_Cyl_W:=G_arrCylinder[_i].stOutput.bWork;

_i:=E_Cylinder.OpenLockRotate;
G_arrCylinder[_i].stInput.bHome:=GVL.I.bOpenLockRotate_Cyl_H;
G_arrCylinder[_i].stInput.bWork:=GVL.I.bOpenLockRotate_Cyl_W;
GVL.Q.bOpenLockRotate_Cyl_H:=G_arrCylinder[_i].stOutput.bHome;
GVL.Q.bOpenLockRotate_Cyl_W:=G_arrCylinder[_i].stOutput.bWork;

_i:=E_Cylinder.OpenLockPush2;
//G_arrCylinder[_i].stInput.bHome:=GVL.I.bOpenLockPush2_Cyl_H;
G_arrCylinder[_i].stInput.bHome:=NOT GVL.I.bOpenLockPush2_Cyl_W;
G_arrCylinder[_i].stInput.bWork:=GVL.I.bOpenLockPush2_Cyl_W;
GVL.Q.bOpenLockPush2_Cyl_H:=G_arrCylinder[_i].stOutput.bHome;
GVL.Q.bOpenLockPush2_Cyl_W:=G_arrCylinder[_i].stOutput.bWork;

_i:=E_Cylinder.TakeUcPrevent;
G_arrCylinder[_i].stInput.bWork:=GVL.I.bTakeUcPrevent_Cyl_W;
GVL.Q.bTakeUcPrevent_Cyl_H:=G_arrCylinder[_i].stOutput.bHome;
GVL.Q.bTakeUcPrevent_Cyl_W:=G_arrCylinder[_i].stOutput.bWork;

_i:=E_Cylinder.TakeUcLift;
G_arrCylinder[_i].stInput.bHome:=GVL.I.bTakeUcLift_Cyl_H;
G_arrCylinder[_i].stInput.bWork:=GVL.I.bTakeUcLift_Cyl_W;
GVL.Q.bTakeUcLift_Cyl_H:=G_arrCylinder[_i].stOutput.bHome;
GVL.Q.bTakeUcLift_Cyl_W:=G_arrCylinder[_i].stOutput.bWork;

_i:=E_Cylinder.TakeUcPush;
G_arrCylinder[_i].stInput.bHome:=GVL.I.bTakeUcPush_Cyl_H;
G_arrCylinder[_i].stInput.bWork:=GVL.I.bTakeUcPush_Cyl_W;
GVL.Q.bTakeUcPush_Cyl_H:=G_arrCylinder[_i].stOutput.bHome;
GVL.Q.bTakeUcPush_Cyl_W:=G_arrCylinder[_i].stOutput.bWork;

_i:=E_Cylinder.TakeUcRotate;
G_arrCylinder[_i].stInput.bHome:=GVL.I.bTakeUcRotate_Cyl_H;
G_arrCylinder[_i].stInput.bWork:=GVL.I.bTakeUcRotate_Cyl_W;
GVL.Q.bTakeUcRotate_Cyl_H:=G_arrCylinder[_i].stOutput.bHome;
GVL.Q.bTakeUcRotate_Cyl_W:=G_arrCylinder[_i].stOutput.bWork;

_i:=E_Cylinder.TakeUcStandard;
G_arrCylinder[_i].stInput.bHome:=GVL.I.bTakeUcStandard_Cyl_H;
G_arrCylinder[_i].stInput.bWork:=GVL.I.bTakeUcStandard_Cyl_W;
GVL.Q.bTakeUcStandard_Cyl_H:=G_arrCylinder[_i].stOutput.bHome;
GVL.Q.bTakeUcStandard_Cyl_W:=G_arrCylinder[_i].stOutput.bWork;

_i:=E_Cylinder.UnloadFrockPrevent;
G_arrCylinder[_i].stInput.bWork:=GVL.I.bUnloadFrockPrevent_Cyl_W;
GVL.Q.bUnloadFrockPrevent_Cyl_H:=G_arrCylinder[_i].stOutput.bHome;
GVL.Q.bUnloadFrockPrevent_Cyl_W:=G_arrCylinder[_i].stOutput.bWork;

_i:=E_Cylinder.UnloadFrockLift;
G_arrCylinder[_i].stInput.bHome:=GVL.I.bUnloadFrockLift_Cyl_H;
G_arrCylinder[_i].stInput.bWork:=GVL.I.bUnloadFrockLift_Cyl_W;
GVL.Q.bUnloadFrockLift_Cyl_H:=G_arrCylinder[_i].stOutput.bHome;
GVL.Q.bUnloadFrockLift_Cyl_W:=G_arrCylinder[_i].stOutput.bWork;

_i:=E_Cylinder.UnloadFrockPush;//
G_arrCylinder[_i].stInput.bHome:=GVL.I.bUnloadFrockPush_Cyl_H;
G_arrCylinder[_i].stInput.bWork:=GVL.I.bUnloadFrockPush_Cyl_W;
GVL.Q.bUnloadFrockPush_Cyl_H:=G_arrCylinder[_i].stOutput.bHome;
GVL.Q.bUnloadFrockPush_Cyl_W:=G_arrCylinder[_i].stOutput.bWork;

_i:=E_Cylinder.TakeUc1Y;
G_arrCylinder[_i].stInput.bHome:=GVL.I.bTakeUc1Y_Cyl_H;
G_arrCylinder[_i].stInput.bWork:=GVL.I.bTakeUc1Y_Cyl_W;
GVL.Q.bTakeUc1Y_Cyl_H:=G_arrCylinder[_i].stOutput.bHome;
GVL.Q.bTakeUc1Y_Cyl_W:=G_arrCylinder[_i].stOutput.bWork;

_i:=E_Cylinder.TakeUc1Z1;
G_arrCylinder[_i].stInput.bHome:=GVL.I.bTakeUc1Z1_Cyl_H;
G_arrCylinder[_i].stInput.bWork:=GVL.I.bTakeUc1Z1_Cyl_W;
GVL.Q.bTakeUc1Z1_Cyl_H:=G_arrCylinder[_i].stOutput.bHome;
GVL.Q.bTakeUc1Z1_Cyl_W:=G_arrCylinder[_i].stOutput.bWork;

_i:=E_Cylinder.TakeUc1Z2;
G_arrCylinder[_i].stInput.bHome:=GVL.I.bTakeUc1Z2_Cyl_H;
G_arrCylinder[_i].stInput.bWork:=GVL.I.bTakeUc1Z2_Cyl_W;
GVL.Q.bTakeUc1Z2_Cyl_H:=G_arrCylinder[_i].stOutput.bHome;
GVL.Q.bTakeUc1Z2_Cyl_W:=G_arrCylinder[_i].stOutput.bWork;

_i:=E_Cylinder.TakeUc1Rotate;
G_arrCylinder[_i].stInput.bHome:=GVL.I.bTakeUc1Rotate_Cyl_H;
G_arrCylinder[_i].stInput.bWork:=GVL.I.bTakeUc1Rotate_Cyl_W;
GVL.Q.bTakeUc1Rotate_Cyl_H:=G_arrCylinder[_i].stOutput.bHome;
GVL.Q.bTakeUc1Rotate_Cyl_W:=G_arrCylinder[_i].stOutput.bWork;

_i:=E_Cylinder.TakeUc1Clamp;
G_arrCylinder[_i].stInput.bHome:=GVL.I.bTakeUc1Clamp_Cyl_H;
//G_arrCylinder[_i].stInput.bWork:=GVL.I.bTakeUc1Clamp_Cyl_W;
GVL.Q.bTakeUc1Clamp_Cyl_H:=G_arrCylinder[_i].stOutput.bHome;
GVL.Q.bTakeUc1Clamp_Cyl_W:=G_arrCylinder[_i].stOutput.bWork;

_i:=E_Cylinder.UnloadUcElevator;
//G_arrCylinder[_i].stInput.bHome:=G_arrCylinder[_i].stOutput.bHome;
//G_arrCylinder[_i].stInput.bWork:=G_arrCylinder[_i].stOutput.bWork;
G_arrCylinder[_i].stInput.bHome:=GVL.I.bUnloadUcElevator_Cyl_H;
G_arrCylinder[_i].stInput.bWork:=GVL.I.bUnloadUcElevator_Cyl_W;
GVL.Q.bUnloadUcElevator_Cyl_H:=G_arrCylinder[_i].stOutput.bHome;
GVL.Q.bUnloadUcElevator_Cyl_W:=G_arrCylinder[_i].stOutput.bWork;

_i:=E_Cylinder.UnloadUcConveyorPush;
//G_arrCylinder[_i].stInput.bHome:=G_arrCylinder[_i].stOutput.bHome;
//G_arrCylinder[_i].stInput.bWork:=G_arrCylinder[_i].stOutput.bWork;
G_arrCylinder[_i].stInput.bHome:=GVL.I.bUnloadUcConveyorPush_Cyl_H;
G_arrCylinder[_i].stInput.bWork:=GVL.I.bUnloadUcConveyorPush_Cyl_W;
GVL.Q.bUnloadUcConveyorPush_Cyl_H:=G_arrCylinder[_i].stOutput.bHome;
GVL.Q.bUnloadUcConveyorPush_Cyl_W:=G_arrCylinder[_i].stOutput.bWork;

_i:=E_Cylinder.UnloadFrockConveyorPrevent;
//G_arrCylinder[_i].stInput.bHome:=G_arrCylinder[_i].stOutput.bHome;
//G_arrCylinder[_i].stInput.bWork:=G_arrCylinder[_i].stOutput.bWork;
G_arrCylinder[_i].stInput.bHome:=GVL.I.bUnloadFrockConveyorPrevent_Cyl_H;
G_arrCylinder[_i].stInput.bWork:=GVL.I.bUnloadFrockConveyorPrevent_Cyl_W;
GVL.Q.bUnloadFrockConveyorPrevent_Cyl_H:=G_arrCylinder[_i].stOutput.bHome;
GVL.Q.bUnloadFrockConveyorPrevent_Cyl_W:=G_arrCylinder[_i].stOutput.bWork;

_i:=E_Cylinder.UnloadFrockConveyorPush;
//G_arrCylinder[_i].stInput.bHome:=G_arrCylinder[_i].stOutput.bHome;
//G_arrCylinder[_i].stInput.bWork:=G_arrCylinder[_i].stOutput.bWork;
G_arrCylinder[_i].stInput.bHome:=GVL.I.bUnloadFrockConveyorPush_Cyl_H;
G_arrCylinder[_i].stInput.bWork:=GVL.I.bUnloadFrockConveyorPush_Cyl_W;
GVL.Q.bUnloadFrockConveyorPush_Cyl_H:=G_arrCylinder[_i].stOutput.bHome;
GVL.Q.bUnloadFrockConveyorPush_Cyl_W:=G_arrCylinder[_i].stOutput.bWork;

_i:=E_Cylinder.OpenLockElevator;
G_arrCylinder[_i].stInput.bHome:=GVL.I.bOpenLockElevator_Cyl_H;
G_arrCylinder[_i].stInput.bWork:=GVL.I.bOpenLockElevator_Cyl_W;
GVL.Q.bOpenLockElevator_Cyl_H:=G_arrCylinder[_i].stOutput.bHome;
GVL.Q.bOpenLockElevator_Cyl_W:=G_arrCylinder[_i].stOutput.bWork;

_i:=E_Cylinder.OpenLockPin;
G_arrCylinder[_i].stInput.bHome:=GVL.I.bOpenLockPin_Cyl_H;
G_arrCylinder[_i].stInput.bWork:=GVL.I.bOpenLockPin_Cyl_W;
GVL.Q.bOpenLockPin_Cyl_H:=G_arrCylinder[_i].stOutput.bHome;
GVL.Q.bOpenLockPin_Cyl_W:=G_arrCylinder[_i].stOutput.bWork;

_i:=E_Cylinder.TakeUcElevator;
G_arrCylinder[_i].stInput.bHome:=GVL.I.bTakeUcElevator_Cyl_H;
G_arrCylinder[_i].stInput.bWork:=GVL.I.bTakeUcElevator_Cyl_W;
GVL.Q.bTakeUcElevator_Cyl_H:=G_arrCylinder[_i].stOutput.bHome;
GVL.Q.bTakeUcElevator_Cyl_W:=G_arrCylinder[_i].stOutput.bWork;

_i:=E_Cylinder.TakeUcPush1;
G_arrCylinder[_i].stInput.bHome:=GVL.I.bTakeUcPush1_Cyl_H;
G_arrCylinder[_i].stInput.bWork:=GVL.I.bTakeUcPush1_Cyl_W;
GVL.Q.bTakeUcPush1_Cyl_H:=G_arrCylinder[_i].stOutput.bHome;
GVL.Q.bTakeUcPush1_Cyl_W:=G_arrCylinder[_i].stOutput.bWork;

_i:=E_Cylinder.UnloadUcBeltTipper;
//G_arrCylinder[_i].stInput.bHome:=GVL.I.bUnloadUcBeltTipper_Cyl_H;
//G_arrCylinder[_i].stInput.bWork:=GVL.I.bUnloadUcBeltTipper_Cyl_W;
GVL.Q.bUnloadUcBeltTipper_Cyl_H:=G_arrCylinder[_i].stOutput.bHome;
GVL.Q.bUnloadUcBeltTipper_Cyl_W:=G_arrCylinder[_i].stOutput.bWork;

_i:=E_Cylinder.UnloadUcBeltLift;
G_arrCylinder[_i].stInput.bHome:=GVL.I.bUnloadUcBeltLift_Cyl_H;
G_arrCylinder[_i].stInput.bWork:=GVL.I.bUnloadUcBeltLift_Cyl_W;
GVL.Q.bUnloadUcBeltLift_Cyl_H:=G_arrCylinder[_i].stOutput.bHome;
GVL.Q.bUnloadUcBeltLift_Cyl_W:=G_arrCylinder[_i].stOutput.bWork;

_i:=E_Cylinder.OpenLockTranslation;
//G_arrCylinder[_i].stInput.bHome:=G_arrCylinder[_i].stOutput.bHome;
//G_arrCylinder[_i].stInput.bWork:=G_arrCylinder[_i].stOutput.bWork;
GVL.Q.bOpenLockTranslation_Cyl_H:=G_arrCylinder[_i].stOutput.bHome;
GVL.Q.bOpenLockTranslation_Cyl_W:=G_arrCylinder[_i].stOutput.bWork;

_i:=E_Cylinder.TakeUcFrockClamp;
G_arrCylinder[_i].stInput.bHome:=GVL.I.bTakeUcFrockClamp_Cyl_H;
G_arrCylinder[_i].stInput.bWork:=GVL.I.bTakeUcFrockClamp_Cyl_W;
GVL.Q.bTakeUcFrockClamp_Cyl_H:=G_arrCylinder[_i].stOutput.bHome;
GVL.Q.bTakeUcFrockClamp_Cyl_W:=G_arrCylinder[_i].stOutput.bWork;
END_ACTION

ACTION A_CylinderTest311:
FOR _i:=0 TO 50 BY 1 DO
	G_arrCylinder[_i].ID:=TO_BYTE(_i+50);
	_arrCylTon_H[_i](IN:=G_arrCylinder[_i].stOutput.bHome , PT:=T#2S , Q=> , ET=> );
	_arrCylTon_W[_i](IN:=G_arrCylinder[_i].stOutput.bWork , PT:=T#2S , Q=> , ET=> );
	G_arrCylinder[_i].stInput.bHome:=_arrCylTon_H[_i].Q;
	G_arrCylinder[_i].stInput.bWork:=_arrCylTon_W[_i].Q;
END_FOR

_i:=E_Cylinder.Line0Part;
GVL.Q.bLine0Part_Cyl_H:=G_arrCylinder[_i].stOutput.bHome;
GVL.Q.bLine0Part_Cyl_W:=G_arrCylinder[_i].stOutput.bWork;

_i:=E_Cylinder.Line0Prevent;
GVL.Q.bLine0Prevent_Cyl_H:=G_arrCylinder[_i].stOutput.bHome;
GVL.Q.bLine0Prevent_Cyl_W:=G_arrCylinder[_i].stOutput.bWork;

_i:=E_Cylinder.Line0Push;
GVL.Q.bLine0Push_Cyl_H:=G_arrCylinder[_i].stOutput.bHome;
GVL.Q.bLine0Push_Cyl_W:=G_arrCylinder[_i].stOutput.bWork;

_i:=E_Cylinder.AcquirePrevent0;
G_arrCylinder[_i].stInput.bWork:=GVL.I.bAcquirePrevent0_Cyl_W;
GVL.Q.bAcquirePrevent0_Cyl_H:=G_arrCylinder[_i].stOutput.bHome;
GVL.Q.bAcquirePrevent0_Cyl_W:=G_arrCylinder[_i].stOutput.bWork;

_i:=E_Cylinder.AcquirePrevent1;
G_arrCylinder[_i].stInput.bWork:=GVL.I.bAcquirePrevent1_Cyl_W;
GVL.Q.bAcquirePrevent1_Cyl_H:=G_arrCylinder[_i].stOutput.bHome;
GVL.Q.bAcquirePrevent1_Cyl_W:=G_arrCylinder[_i].stOutput.bWork;

_i:=E_Cylinder.AcquireLift;
G_arrCylinder[_i].stInput.bHome:=GVL.I.bAcquireLift_Cyl_H;
G_arrCylinder[_i].stInput.bWork:=GVL.I.bAcquireLift_Cyl_W;
GVL.Q.bAcquireLift_Cyl_H:=G_arrCylinder[_i].stOutput.bHome;
GVL.Q.bAcquireLift_Cyl_W:=G_arrCylinder[_i].stOutput.bWork;

_i:=E_Cylinder.AcquirePush;
G_arrCylinder[_i].stInput.bHome:=GVL.I.bAcquirePush_Cyl_H;
G_arrCylinder[_i].stInput.bWork:=GVL.I.bAcquirePush_Cyl_W;
GVL.Q.bAcquirePush_Cyl_H:=G_arrCylinder[_i].stOutput.bHome;
GVL.Q.bAcquirePush_Cyl_W:=G_arrCylinder[_i].stOutput.bWork;

_i:=E_Cylinder.AcquireElevator;
G_arrCylinder[_i].stInput.bHome:=GVL.I.bAcquireElevator_Cyl_H;
G_arrCylinder[_i].stInput.bWork:=GVL.I.bAcquireElevator_Cyl_W;
GVL.Q.bAcquireElevator_Cyl_H:=G_arrCylinder[_i].stOutput.bHome;
GVL.Q.bAcquireElevator_Cyl_W:=G_arrCylinder[_i].stOutput.bWork;

_i:=E_Cylinder.SteeringLift;
G_arrCylinder[_i].stInput.bHome:=GVL.I.bSteeringLift_Cyl_H;
G_arrCylinder[_i].stInput.bWork:=GVL.I.bSteeringLift_Cyl_W;
GVL.Q.bSteeringLift_Cyl_H:=G_arrCylinder[_i].stOutput.bHome;
GVL.Q.bSteeringLift_Cyl_W:=G_arrCylinder[_i].stOutput.bWork;

_i:=E_Cylinder.SteeringAcquireElevator;
G_arrCylinder[_i].stInput.bHome:=GVL.I.bSteeringAcquireElevator_Cyl_H;
G_arrCylinder[_i].stInput.bWork:=GVL.I.bSteeringAcquireElevator_Cyl_W;
GVL.Q.bSteeringAcquireElevator_Cyl_H:=G_arrCylinder[_i].stOutput.bHome;
GVL.Q.bSteeringAcquireElevator_Cyl_W:=G_arrCylinder[_i].stOutput.bWork;

_i:=E_Cylinder.SteeringRotate;
//G_arrCylinder[_i].stInput.bHome:=GVL.I.bSteeringRotate_Cyl_H;
G_arrCylinder[_i].stInput.bWork:=GVL.I.bSteeringRotate_Cyl_W;
GVL.Q.bSteeringRotate_Cyl_H:=G_arrCylinder[_i].stOutput.bHome;
GVL.Q.bSteeringRotate_Cyl_W:=G_arrCylinder[_i].stOutput.bWork;

_i:=E_Cylinder.SteeringAcquireLimit;
G_arrCylinder[_i].stInput.bHome:=GVL.I.bSteeringAcquireLimit_Cyl_H;
//G_arrCylinder[_i].stInput.bWork:=GVL.I.bSteeringAcquireLimit_Cyl_W;
GVL.Q.bSteeringAcquireLimit_Cyl_H:=G_arrCylinder[_i].stOutput.bHome;
GVL.Q.bSteeringAcquireLimit_Cyl_W:=G_arrCylinder[_i].stOutput.bWork;

_i:=E_Cylinder.OpenLockPrevent;
G_arrCylinder[_i].stInput.bWork:=GVL.I.bOpenLockPrevent_Cyl_W;
GVL.Q.bOpenLockPrevent_Cyl_H:=G_arrCylinder[_i].stOutput.bHome;
GVL.Q.bOpenLockPrevent_Cyl_W:=G_arrCylinder[_i].stOutput.bWork;

_i:=E_Cylinder.OpenLockLift;
G_arrCylinder[_i].stInput.bHome:=GVL.I.bOpenLockLift_Cyl_H;
G_arrCylinder[_i].stInput.bWork:=GVL.I.bOpenLockLift_Cyl_W;
GVL.Q.bOpenLockLift_Cyl_H:=G_arrCylinder[_i].stOutput.bHome;
GVL.Q.bOpenLockLift_Cyl_W:=G_arrCylinder[_i].stOutput.bWork;

